LIN {X 0,Y 327.842,Z 1176.159,A -85,B 0,C 180,E1 13690.608,E2 13690.608} C_VEL
LIN {X 0,Y 330.278,Z 1159.38,A -85,B 0,C 180,E1 13695.569,E2 13695.569} C_VEL
LIN {X 0,Y 333.559,Z 1138.416,A -85,B 0,C 180,E1 13699.833,E2 13699.833} C_VEL
LIN {X 0,Y 337.656,Z 1111.754,A -85,B 0,C 180,E1 13703.592,E2 13703.592} C_VEL
LIN {X 0,Y 341.285,Z 1081.785,A -85,B 0,C 180,E1 13706.42,E2 13706.42} C_VEL
LIN {X 0,Y 343.694,Z 1048.536,A -85,B 0,C 180,E1 13708.37,E2 13708.37} C_VEL
LIN {X 0,Y 324.455,Z 997.109,A -85,B 0,C 180,E1 13712.143,E2 13712.143} C_VEL
LIN {X 0,Y 321.566,Z 989.03,A -85,B 0,C 180,E1 13712.907,E2 13712.907} C_VEL
LIN {X 0,Y 321.361,Z 989.03,A -85,B 0,C 180,E1 13715.329,E2 13715.329} C_VEL
LIN {X 0,Y 323.535,Z 994.456,A -85,B 0,C 180,E1 13716.08,E2 13716.08} C_VEL
LIN {X 0,Y 326.454,Z 998.467,A -85,B 0,C 180,E1 13716.933,E2 13716.933} C_VEL
LIN {X 0,Y 341.328,Z 1021.069,A -85,B 0,C 180,E1 13720.903,E2 13720.903} C_VEL
LIN {X 0,Y 357.405,Z 1050.395,A -85,B 0,C 180,E1 13724.791,E2 13724.791} C_VEL
LIN {X 0,Y 367.108,Z 1076.272,A -85,B 0,C 180,E1 13727.719,E2 13727.719} C_VEL
LIN {X 0,Y 361.475,Z 1112.177,A -85,B 0,C 180,E1 13729.868,E2 13729.868} C_VEL
LIN {X 0,Y 354.22,Z 1145.406,A -85,B 0,C 180,E1 13732.909,E2 13732.909} C_VEL
LIN {X 0,Y 346.259,Z 1175.129,A -85,B 0,C 180,E1 13736.799,E2 13736.799} C_VEL
LIN {X 0,Y 338.326,Z 1201.655,A -85,B 0,C 180,E1 13741.706,E2 13741.706} C_VEL
LIN {X 0,Y 331.825,Z 1222.692,A -85,B 0,C 180,E1 13747.254,E2 13747.254} C_VEL
LIN {X 0,Y 327.378,Z 1238.391,A -85,B 0,C 180,E1 13753.251,E2 13753.251} C_VEL
LIN {X 0,Y 325.075,Z 1248.624,A -85,B 0,C 180,E1 13759.294,E2 13759.294} C_VEL
LIN {X 0,Y 324.228,Z 1253.714,A -85,B 0,C 180,E1 13764.654,E2 13764.654} C_VEL
LIN {X 0,Y 323.952,Z 1255.427,A -85,B 0,C 180,E1 13769.995,E2 13769.995} C_VEL
LIN {X 0,Y 324.317,Z 1252.709,A -85,B 0,C 180,E1 13776.675,E2 13776.675} C_VEL
LIN {X 0,Y 325.921,Z 1244.536,A -85,B 0,C 180,E1 13783.38,E2 13783.38} C_VEL
LIN {X 0,Y 329.451,Z 1230.706,A -85,B 0,C 180,E1 13789.903,E2 13789.903} C_VEL
LIN {X 0,Y 335.08,Z 1211.817,A -85,B 0,C 180,E1 13795.758,E2 13795.758} C_VEL
LIN {X 0,Y 342.404,Z 1188.224,A -85,B 0,C 180,E1 13800.886,E2 13800.886} C_VEL
LIN {X 0,Y 350.57,Z 1159.61,A -85,B 0,C 180,E1 13805.301,E2 13805.301} C_VEL
LIN {X 0,Y 358.19,Z 1128.049,A -85,B 0,C 180,E1 13808.714,E2 13808.714} C_VEL
LIN {X 0,Y 364.641,Z 1093.639,A -85,B 0,C 180,E1 13811.261,E2 13811.261} C_VEL
LIN {X 0,Y 366.791,Z 1074.45,A -85,B 0,C 180,E1 13812.336,E2 13812.336} C_VEL
LIN {X 0,Y 354.759,Z 1045.172,A -85,B 0,C 180,E1 13815.748,E2 13815.748} C_VEL
LIN {X 0,Y 336.902,Z 1013.596,A -85,B 0,C 180,E1 13820.109,E2 13820.109} C_VEL
LIN {X 0,Y 323.813,Z 994.624,A -85,B 0,C 180,E1 13823.712,E2 13823.712} C_VEL
LIN {X 0,Y 321.462,Z 989.03,A -85,B 0,C 180,E1 13824.571,E2 13824.571} C_VEL
LIN {X 0,Y 321.795,Z 989.03,A -85,B 0,C 180,E1 13832.988,E2 13832.988} C_VEL
LIN {X 0,Y 322.198,Z 989.03,A -85,B 0,C 180,E1 13840.864,E2 13840.864} C_VEL
LIN {X 0,Y 322.712,Z 989.03,A -85,B 0,C 180,E1 13849.083,E2 13849.083} C_VEL
LIN {X 0,Y 323.215,Z 989.03,A -85,B 0,C 180,E1 13857.325,E2 13857.325} C_VEL
LIN {X 0,Y 323.277,Z 989.03,A -85,B 0,C 180,E1 13862.676,E2 13862.676} C_VEL
LIN {X 0,Y 322.641,Z 989.03,A -85,B 0,C 180,E1 13870.851,E2 13870.851} C_VEL
LIN {X 0,Y 322.111,Z 989.03,A -85,B 0,C 180,E1 13879.143,E2 13879.143} C_VEL
LIN {X 0,Y 321.771,Z 989.03,A -85,B 0,C 180,E1 13887.003,E2 13887.003} C_VEL
LIN {X 0,Y 321.635,Z 989.591,A -85,B 0,C 180,E1 13892.594,E2 13892.594} C_VEL
LIN {X 0,Y 326.494,Z 1001.003,A -85,B 0,C 180,E1 13894.238,E2 13894.238} C_VEL
LIN {X 0,Y 349.905,Z 1049.922,A -85,B 0,C 180,E1 13899.619,E2 13899.619} C_VEL
LIN {X 0,Y 364.312,Z 1087.174,A -85,B 0,C 180,E1 13903.441,E2 13903.441} C_VEL
LIN {X 0,Y 365.005,Z 1093.61,A -85,B 0,C 180,E1 13903.961,E2 13903.961} C_VEL
LIN {X 0,Y 357.243,Z 1134.418,A -85,B 0,C 180,E1 13906.643,E2 13906.643} C_VEL
LIN {X 0,Y 348.266,Z 1174.72,A -85,B 0,C 180,E1 13910.507,E2 13910.507} C_VEL
LIN {X 0,Y 340.072,Z 1213.611,A -85,B 0,C 180,E1 13915.375,E2 13915.375} C_VEL
LIN {X 0,Y 333.762,Z 1242.406,A -85,B 0,C 180,E1 13920.448,E2 13920.448} C_VEL
LIN {X 0,Y 328.614,Z 1266.532,A -85,B 0,C 180,E1 13926.32,E2 13926.32} C_VEL
LIN {X 0,Y 325.489,Z 1284.698,A -85,B 0,C 180,E1 13932.645,E2 13932.645} C_VEL
LIN {X 0,Y 324.33,Z 1296.014,A -85,B 0,C 180,E1 13938.468,E2 13938.468} C_VEL
LIN {X 0,Y 323.881,Z 1302.925,A -85,B 0,C 180,E1 13944.658,E2 13944.658} C_VEL
LIN {X 0,Y 323.958,Z 1304.876,A -85,B 0,C 180,E1 13950.005,E2 13950.005} C_VEL
LIN {X 0,Y 323.912,Z 1302.924,A -85,B 0,C 180,E1 13955.352,E2 13955.352} C_VEL
LIN {X 0,Y 324.362,Z 1295.959,A -85,B 0,C 180,E1 13961.572,E2 13961.572} C_VEL
LIN {X 0,Y 325.988,Z 1282.805,A -85,B 0,C 180,E1 13968.159,E2 13968.159} C_VEL
LIN {X 0,Y 329.344,Z 1264.057,A -85,B 0,C 180,E1 13974.36,E2 13974.36} C_VEL
LIN {X 0,Y 334.543,Z 1240.153,A -85,B 0,C 180,E1 13980.001,E2 13980.001} C_VEL
LIN {X 0,Y 338.144,Z 1224.571,A -85,B 0,C 180,E1 13982.848,E2 13982.848} C_VEL
LIN {X 0,Y 337.312,Z 1212.87,A -85,B 0,C 180,E1 13985.069,E2 13985.069} C_VEL
LIN {X 0,Y 336.399,Z 1202.111,A -85,B 0,C 180,E1 13986.93,E2 13986.93} C_VEL
LIN {X 0,Y 336.725,Z 1200.392,A -85,B 0,C 180,E1 13987.157,E2 13987.157} C_VEL
LIN {X 0,Y 343.446,Z 1167.637,A -85,B 0,C 180,E1 13990.804,E2 13990.804} C_VEL
LIN {X 0,Y 350.339,Z 1129.054,A -85,B 0,C 180,E1 13993.983,E2 13993.983} C_VEL
LIN {X 0,Y 360.86,Z 1090.849,A -85,B 0,C 180,E1 13997.195,E2 13997.195} C_VEL
LIN {X 0,Y 364.072,Z 1066.549,A -85,B 0,C 180,E1 14000.478,E2 14000.478} C_VEL
LIN {X 0,Y 363.409,Z 1063.296,A -85,B 0,C 180,E1 14002.097,E2 14002.097} C_VEL
LIN {X 0,Y 362.843,Z 1064.438,A -85,B 0,C 180,E1 14004.393,E2 14004.393} C_VEL
LIN {X 0,Y 359.681,Z 1073.138,A -85,B 0,C 180,E1 14005.221,E2 14005.221} C_VEL
LIN {X 0,Y 348.848,Z 1111.499,A -85,B 0,C 180,E1 14008.576,E2 14008.576} C_VEL
LIN {X 0,Y 341.201,Z 1138.326,A -85,B 0,C 180,E1 14012.044,E2 14012.044} C_VEL
LIN {X 0,Y 333.916,Z 1160.821,A -85,B 0,C 180,E1 14016.355,E2 14016.355} C_VEL
LIN {X 0,Y 327.641,Z 1177.723,A -85,B 0,C 180,E1 14021.192,E2 14021.192} C_VEL
LIN {X 0,Y 323.111,Z 1189.142,A -85,B 0,C 180,E1 14026.496,E2 14026.496} C_VEL
LIN {X 0,Y 320.196,Z 1195.188,A -85,B 0,C 180,E1 14031.872,E2 14031.872} C_VEL
LIN {X 0,Y 318.796,Z 1196.308,A -85,B 0,C 180,E1 14037.287,E2 14037.287} C_VEL
LIN {X 0,Y 318.677,Z 1192.532,A -85,B 0,C 180,E1 14042.713,E2 14042.713} C_VEL
LIN {X 0,Y 319.227,Z 1183.709,A -85,B 0,C 180,E1 14048.152,E2 14048.152} C_VEL
LIN {X 0,Y 321.312,Z 1168.881,A -85,B 0,C 180,E1 14053.58,E2 14053.58} C_VEL
LIN {X 0,Y 324.532,Z 1148.483,A -85,B 0,C 180,E1 14058.523,E2 14058.523} C_VEL
LIN {X 0,Y 328.668,Z 1122.896,A -85,B 0,C 180,E1 14062.74,E2 14062.74} C_VEL
LIN {X 0,Y 332.615,Z 1094.968,A -85,B 0,C 180,E1 14065.89,E2 14065.89} C_VEL
LIN {X 0,Y 335.845,Z 1063.866,A -85,B 0,C 180,E1 14068.183,E2 14068.183} C_VEL
LIN {X 0,Y 336.162,Z 1049.341,A -85,B 0,C 180,E1 14068.96,E2 14068.96} C_VEL
LIN {X 0,Y 316.792,Z 997.606,A -85,B 0,C 180,E1 14072.918,E2 14072.918} C_VEL
LIN {X 0,Y 314.162,Z 991.943,A -85,B 0,C 180,E1 14073.524,E2 14073.524} C_VEL
LIN {X 0,Y 318.931,Z 999.004,A -85,B 0,C 180,E1 14075.089,E2 14075.089} C_VEL
LIN {X 0,Y 333.802,Z 1021.018,A -85,B 0,C 180,E1 14079.365,E2 14079.365} C_VEL
LIN {X 0,Y 350.514,Z 1050.918,A -85,B 0,C 180,E1 14083.64,E2 14083.64} C_VEL
LIN {X 0,Y 361.022,Z 1078.194,A -85,B 0,C 180,E1 14086.924,E2 14086.924} C_VEL
LIN {X 0,Y 355.102,Z 1114.621,A -85,B 0,C 180,E1 14089.197,E2 14089.197} C_VEL
LIN {X 0,Y 347.376,Z 1148.214,A -85,B 0,C 180,E1 14092.376,E2 14092.376} C_VEL
LIN {X 0,Y 338.737,Z 1178.747,A -85,B 0,C 180,E1 14096.538,E2 14096.538} C_VEL
LIN {X 0,Y 330.839,Z 1203.66,A -85,B 0,C 180,E1 14101.378,E2 14101.378} C_VEL
LIN {X 0,Y 324.163,Z 1224.334,A -85,B 0,C 180,E1 14107.048,E2 14107.048} C_VEL
LIN {X 0,Y 319.393,Z 1240.43,A -85,B 0,C 180,E1 14113.526,E2 14113.526} C_VEL
LIN {X 0,Y 316.955,Z 1250.823,A -85,B 0,C 180,E1 14120.402,E2 14120.402} C_VEL
LIN {X 0,Y 316.173,Z 1255.575,A -85,B 0,C 180,E1 14127.259,E2 14127.259} C_VEL
LIN {X 0,Y 316.198,Z 1255.54,A -85,B 0,C 180,E1 14132.73,E2 14132.73} C_VEL
LIN {X 0,Y 316.945,Z 1250.727,A -85,B 0,C 180,E1 14139.587,E2 14139.587} C_VEL
LIN {X 0,Y 319.447,Z 1240.258,A -85,B 0,C 180,E1 14146.46,E2 14146.46} C_VEL
LIN {X 0,Y 324.215,Z 1224.067,A -85,B 0,C 180,E1 14152.937,E2 14152.937} C_VEL
LIN {X 0,Y 330.892,Z 1203.309,A -85,B 0,C 180,E1 14158.605,E2 14158.605} C_VEL
LIN {X 0,Y 339.197,Z 1177.241,A -85,B 0,C 180,E1 14163.59,E2 14163.59} C_VEL
LIN {X 0,Y 347.536,Z 1147.512,A -85,B 0,C 180,E1 14167.597,E2 14167.597} C_VEL
LIN {X 0,Y 354.85,Z 1115.563,A -85,B 0,C 180,E1 14170.625,E2 14170.625} C_VEL
LIN {X 0,Y 360.985,Z 1078.194,A -85,B 0,C 180,E1 14172.972,E2 14172.972} C_VEL
LIN {X 0,Y 349.196,Z 1048.427,A -85,B 0,C 180,E1 14176.591,E2 14176.591} C_VEL
LIN {X 0,Y 332.009,Z 1018.103,A -85,B 0,C 180,E1 14180.992,E2 14180.992} C_VEL
LIN {X 0,Y 316.548,Z 995.18,A -85,B 0,C 180,E1 14185.552,E2 14185.552} C_VEL
LIN {X 0,Y 313.63,Z 990.188,A -85,B 0,C 180,E1 14186.555,E2 14186.555} C_VEL
LIN {X 0,Y 313.543,Z 989.03,A -85,B 0,C 180,E1 14186.73,E2 14186.73} C_VEL
LIN {X 0,Y 313.9,Z 989.03,A -85,B 0,C 180,E1 14194.366,E2 14194.366} C_VEL
LIN {X 0,Y 314.252,Z 989.03,A -85,B 0,C 180,E1 14200.36,E2 14200.36} C_VEL
LIN {X 0,Y 314.623,Z 989.03,A -85,B 0,C 180,E1 14206.126,E2 14206.126} C_VEL
LIN {X 0,Y 315.194,Z 989.03,A -85,B 0,C 180,E1 14214.506,E2 14214.506} C_VEL
LIN {X 0,Y 315.547,Z 989.03,A -85,B 0,C 180,E1 14220.001,E2 14220.001} C_VEL
LIN {X 0,Y 314.913,Z 989.03,A -85,B 0,C 180,E1 14228.265,E2 14228.265} C_VEL
LIN {X 0,Y 314.348,Z 989.03,A -85,B 0,C 180,E1 14236.74,E2 14236.74} C_VEL
LIN {X 0,Y 313.896,Z 989.03,A -85,B 0,C 180,E1 14244.03,E2 14244.03} C_VEL
LIN {X 0,Y 313.713,Z 989.516,A -85,B 0,C 180,E1 14251.427,E2 14251.427} C_VEL
LIN {X 0,Y 321.069,Z 1005.61,A -85,B 0,C 180,E1 14253.62,E2 14253.62} C_VEL
LIN {X 0,Y 342.911,Z 1051.628,A -85,B 0,C 180,E1 14258.834,E2 14258.834} C_VEL
LIN {X 0,Y 357.162,Z 1088.674,A -85,B 0,C 180,E1 14262.792,E2 14262.792} C_VEL
LIN {X 0,Y 358.136,Z 1095.156,A -85,B 0,C 180,E1 14263.365,E2 14263.365} C_VEL
LIN {X 0,Y 350.166,Z 1135.277,A -85,B 0,C 180,E1 14266.092,E2 14266.092} C_VEL
LIN {X 0,Y 338.301,Z 1190.611,A -85,B 0,C 180,E1 14271.565,E2 14271.565} C_VEL
LIN {X 0,Y 331.425,Z 1221.512,A -85,B 0,C 180,E1 14275.929,E2 14275.929} C_VEL
LIN {X 0,Y 324.948,Z 1248.483,A -85,B 0,C 180,E1 14281.203,E2 14281.203} C_VEL
LIN {X 0,Y 320.163,Z 1270.395,A -85,B 0,C 180,E1 14287.128,E2 14287.128} C_VEL
LIN {X 0,Y 317.357,Z 1286.85,A -85,B 0,C 180,E1 14293.428,E2 14293.428} C_VEL
LIN {X 0,Y 316.362,Z 1296.606,A -85,B 0,C 180,E1 14299.006,E2 14299.006} C_VEL
LIN {X 0,Y 316.012,Z 1302.321,A -85,B 0,C 180,E1 14304.525,E2 14304.525} C_VEL
LIN {X 0,Y 316.104,Z 1304.276,A -85,B 0,C 180,E1 14310.005,E2 14310.005} C_VEL
LIN {X 0,Y 316.042,Z 1302.321,A -85,B 0,C 180,E1 14315.485,E2 14315.485} C_VEL
LIN {X 0,Y 316.51,Z 1295.348,A -85,B 0,C 180,E1 14321.863,E2 14321.863} C_VEL
LIN {X 0,Y 318.19,Z 1282.521,A -85,B 0,C 180,E1 14328.475,E2 14328.475} C_VEL
LIN {X 0,Y 321.855,Z 1263.434,A -85,B 0,C 180,E1 14334.965,E2 14334.965} C_VEL
LIN {X 0,Y 327.182,Z 1240.622,A -85,B 0,C 180,E1 14340.493,E2 14340.493} C_VEL
LIN {X 0,Y 333.928,Z 1212.709,A -85,B 0,C 180,E1 14345.43,E2 14345.43} C_VEL
LIN {X 0,Y 336.725,Z 1200.392,A -85,B 0,C 180,E1 14347.157,E2 14347.157} C_VEL
LIN {X 0,Y 336.432,Z 1187.381,A -85,B 0,C 180,E1 14349.14,E2 14349.14} C_VEL
LIN {X 0,Y 336.001,Z 1173.826,A -85,B 0,C 180,E1 14351.05,E2 14351.05} C_VEL
LIN {X 0,Y 343.866,Z 1132.971,A -85,B 0,C 180,E1 14354.607,E2 14354.607} C_VEL
LIN {X 0,Y 356.018,Z 1093.556,A -85,B 0,C 180,E1 14358.141,E2 14358.141} C_VEL
LIN {X 0,Y 360.214,Z 1071.69,A -85,B 0,C 180,E1 14361.386,E2 14361.386} C_VEL
LIN {X 0,Y 359.528,Z 1070.736,A -85,B 0,C 180,E1 14362.899,E2 14362.899} C_VEL
LIN {X 0,Y 358.958,Z 1072.007,A -85,B 0,C 180,E1 14363.79,E2 14363.79} C_VEL
LIN {X 0,Y 346.824,Z 1105.191,A -85,B 0,C 180,E1 14366.682,E2 14366.682} C_VEL
LIN {X 0,Y 337.416,Z 1135.219,A -85,B 0,C 180,E1 14370.348,E2 14370.348} C_VEL
LIN {X 0,Y 329.312,Z 1158.383,A -85,B 0,C 180,E1 14374.559,E2 14374.559} C_VEL
LIN {X 0,Y 321.97,Z 1176.979,A -85,B 0,C 180,E1 14379.632,E2 14379.632} C_VEL
LIN {X 0,Y 316.713,Z 1188.932,A -85,B 0,C 180,E1 14384.808,E2 14384.808} C_VEL
LIN {X 0,Y 313.197,Z 1195.941,A -85,B 0,C 180,E1 14390.292,E2 14390.292} C_VEL
LIN {X 0,Y 311.7,Z 1197.938,A -85,B 0,C 180,E1 14394.443,E2 14394.443} C_VEL
LIN {X 0,Y 310.898,Z 1196.392,A -85,B 0,C 180,E1 14399.999,E2 14399.999} C_VEL
LIN {X 0,Y 311.072,Z 1189.934,A -85,B 0,C 180,E1 14405.567,E2 14405.567} C_VEL
LIN {X 0,Y 312.428,Z 1178.022,A -85,B 0,C 180,E1 14411.138,E2 14411.138} C_VEL
LIN {X 0,Y 315.168,Z 1160.215,A -85,B 0,C 180,E1 14416.483,E2 14416.483} C_VEL
LIN {X 0,Y 319.063,Z 1137.233,A -85,B 0,C 180,E1 14421.137,E2 14421.137} C_VEL
LIN {X 0,Y 323.293,Z 1110.729,A -85,B 0,C 180,E1 14424.838,E2 14424.838} C_VEL
LIN {X 0,Y 327.037,Z 1081.274,A -85,B 0,C 180,E1 14427.627,E2 14427.627} C_VEL
LIN {X 0,Y 329.022,Z 1051.34,A -85,B 0,C 180,E1 14429.465,E2 14429.465} C_VEL
LIN {X 0,Y 311.515,Z 1003.891,A -85,B 0,C 180,E1 14433.272,E2 14433.272} C_VEL
LIN {X 0,Y 315.033,Z 1004.213,A -85,B 0,C 180,E1 14434.262,E2 14434.262} C_VEL
LIN {X 0,Y 331.258,Z 1029.023,A -85,B 0,C 180,E1 14439.092,E2 14439.092} C_VEL
LIN {X 0,Y 346.122,Z 1056.913,A -85,B 0,C 180,E1 14443.149,E2 14443.149} C_VEL
LIN {X 0,Y 355.015,Z 1080.978,A -85,B 0,C 180,E1 14446.161,E2 14446.161} C_VEL
LIN {X 0,Y 348.772,Z 1117.031,A -85,B 0,C 180,E1 14448.5,E2 14448.5} C_VEL
LIN {X 0,Y 340.844,Z 1149.896,A -85,B 0,C 180,E1 14451.69,E2 14451.69} C_VEL
LIN {X 0,Y 332.129,Z 1179.342,A -85,B 0,C 180,E1 14455.781,E2 14455.781} C_VEL
LIN {X 0,Y 323.86,Z 1204.261,A -85,B 0,C 180,E1 14460.702,E2 14460.702} C_VEL
LIN {X 0,Y 316.806,Z 1224.941,A -85,B 0,C 180,E1 14466.483,E2 14466.483} C_VEL
LIN {X 0,Y 311.778,Z 1241.034,A -85,B 0,C 180,E1 14473.112,E2 14473.112} C_VEL
LIN {X 0,Y 309.158,Z 1251.426,A -85,B 0,C 180,E1 14480.158,E2 14480.158} C_VEL
LIN {X 0,Y 308.296,Z 1256.177,A -85,B 0,C 180,E1 14487.189,E2 14487.189} C_VEL
LIN {X 0,Y 308.321,Z 1256.143,A -85,B 0,C 180,E1 14492.8,E2 14492.8} C_VEL
LIN {X 0,Y 309.148,Z 1251.331,A -85,B 0,C 180,E1 14499.832,E2 14499.832} C_VEL
LIN {X 0,Y 311.823,Z 1240.866,A -85,B 0,C 180,E1 14506.874,E2 14506.874} C_VEL
LIN {X 0,Y 316.875,Z 1224.676,A -85,B 0,C 180,E1 14513.5,E2 14513.5} C_VEL
LIN {X 0,Y 323.917,Z 1203.915,A -85,B 0,C 180,E1 14519.28,E2 14519.28} C_VEL
LIN {X 0,Y 332.594,Z 1177.843,A -85,B 0,C 180,E1 14524.349,E2 14524.349} C_VEL
LIN {X 0,Y 340.996,Z 1149.242,A -85,B 0,C 180,E1 14528.278,E2 14528.278} C_VEL
LIN {X 0,Y 348.514,Z 1117.987,A -85,B 0,C 180,E1 14531.318,E2 14531.318} C_VEL
LIN {X 0,Y 354.838,Z 1082.755,A -85,B 0,C 180,E1 14533.623,E2 14533.623} C_VEL
LIN {X 0,Y 350.86,Z 1068.778,A -85,B 0,C 180,E1 14535.233,E2 14535.233} C_VEL
LIN {X 0,Y 337.118,Z 1039.09,A -85,B 0,C 180,E1 14539.23,E2 14539.23} C_VEL
LIN {X 0,Y 321.388,Z 1013.578,A -85,B 0,C 180,E1 14543.601,E2 14543.601} C_VEL
LIN {X 0,Y 308.804,Z 995.31,A -85,B 0,C 180,E1 14547.738,E2 14547.738} C_VEL
LIN {X 0,Y 305.784,Z 990.191,A -85,B 0,C 180,E1 14548.892,E2 14548.892} C_VEL
LIN {X 0,Y 305.682,Z 989.03,A -85,B 0,C 180,E1 14549.13,E2 14549.13} C_VEL
LIN {X 0,Y 306.069,Z 989.03,A -85,B 0,C 180,E1 14556.772,E2 14556.772} C_VEL
LIN {X 0,Y 306.464,Z 989.03,A -85,B 0,C 180,E1 14562.818,E2 14562.818} C_VEL
LIN {X 0,Y 306.878,Z 989.03,A -85,B 0,C 180,E1 14569.544,E2 14569.544} C_VEL
LIN {X 0,Y 307.406,Z 989.03,A -85,B 0,C 180,E1 14577.187,E2 14577.187} C_VEL
LIN {X 0,Y 307.45,Z 989.03,A -85,B 0,C 180,E1 14582.814,E2 14582.814} C_VEL
LIN {X 0,Y 306.79,Z 989.03,A -85,B 0,C 180,E1 14591.347,E2 14591.347} C_VEL
LIN {X 0,Y 306.362,Z 989.03,A -85,B 0,C 180,E1 14597.189,E2 14597.189} C_VEL
LIN {X 0,Y 306.035,Z 989.03,A -85,B 0,C 180,E1 14603.232,E2 14603.232} C_VEL
LIN {X 0,Y 305.787,Z 989.513,A -85,B 0,C 180,E1 14610.217,E2 14610.217} C_VEL
LIN {X 0,Y 331.983,Z 1044.448,A -85,B 0,C 180,E1 14617.031,E2 14617.031} C_VEL
LIN {X 0,Y 347.243,Z 1082.028,A -85,B 0,C 180,E1 14621.241,E2 14621.241} C_VEL
LIN {X 0,Y 351.243,Z 1096.676,A -85,B 0,C 180,E1 14622.751,E2 14622.751} C_VEL
LIN {X 0,Y 342.748,Z 1137.423,A -85,B 0,C 180,E1 14625.652,E2 14625.652} C_VEL
LIN {X 0,Y 333.546,Z 1182.943,A -85,B 0,C 180,E1 14629.863,E2 14629.863} C_VEL
LIN {X 0,Y 325.934,Z 1215.257,A -85,B 0,C 180,E1 14634.194,E2 14634.194} C_VEL
LIN {X 0,Y 318.997,Z 1243.26,A -85,B 0,C 180,E1 14639.439,E2 14639.439} C_VEL
LIN {X 0,Y 313.317,Z 1266.602,A -85,B 0,C 180,E1 14645.534,E2 14645.534} C_VEL
LIN {X 0,Y 309.911,Z 1284.212,A -85,B 0,C 180,E1 14652.087,E2 14652.087} C_VEL
LIN {X 0,Y 308.491,Z 1295.994,A -85,B 0,C 180,E1 14658.722,E2 14658.722} C_VEL
LIN {X 0,Y 308.125,Z 1301.717,A -85,B 0,C 180,E1 14664.384,E2 14664.384} C_VEL
LIN {X 0,Y 308.223,Z 1303.675,A -85,B 0,C 180,E1 14670.005,E2 14670.005} C_VEL
LIN {X 0,Y 308.157,Z 1301.717,A -85,B 0,C 180,E1 14675.626,E2 14675.626} C_VEL
LIN {X 0,Y 308.634,Z 1294.852,A -85,B 0,C 180,E1 14682.088,E2 14682.088} C_VEL
LIN {X 0,Y 310.433,Z 1281.899,A -85,B 0,C 180,E1 14688.954,E2 14688.954} C_VEL
LIN {X 0,Y 314.423,Z 1262.813,A -85,B 0,C 180,E1 14695.597,E2 14695.597} C_VEL
LIN {X 0,Y 320.459,Z 1238.681,A -85,B 0,C 180,E1 14701.523,E2 14701.523} C_VEL
LIN {X 0,Y 328.063,Z 1208.903,A -85,B 0,C 180,E1 14706.732,E2 14706.732} C_VEL
LIN {X 0,Y 335.108,Z 1178.061,A -85,B 0,C 180,E1 14710.602,E2 14710.602} C_VEL
LIN {X 0,Y 336.001,Z 1173.826,A -85,B 0,C 180,E1 14711.05,E2 14711.05} C_VEL
LIN {X 0,Y 335.675,Z 1159.744,A -85,B 0,C 180,E1 14712.836,E2 14712.836} C_VEL
LIN {X 0,Y 335.217,Z 1145.107,A -85,B 0,C 180,E1 14714.475,E2 14714.475} C_VEL
LIN {X 0,Y 351.463,Z 1096.768,A -85,B 0,C 180,E1 14719.077,E2 14719.077} C_VEL
LIN {X 0,Y 356.158,Z 1079.085,A -85,B 0,C 180,E1 14721.765,E2 14721.765} C_VEL
LIN {X 0,Y 356.283,Z 1077.707,A -85,B 0,C 180,E1 14722.503,E2 14722.503} C_VEL
LIN {X 0,Y 355.21,Z 1079.638,A -85,B 0,C 180,E1 14723.024,E2 14723.024} C_VEL
LIN {X 0,Y 341.927,Z 1110.917,A -85,B 0,C 180,E1 14725.95,E2 14725.95} C_VEL
LIN {X 0,Y 331.015,Z 1140.662,A -85,B 0,C 180,E1 14729.904,E2 14729.904} C_VEL
LIN {X 0,Y 322.199,Z 1163.055,A -85,B 0,C 180,E1 14734.329,E2 14734.329} C_VEL
LIN {X 0,Y 314.207,Z 1181.108,A -85,B 0,C 180,E1 14739.732,E2 14739.732} C_VEL
LIN {X 0,Y 308.819,Z 1192.227,A -85,B 0,C 180,E1 14745.136,E2 14745.136} C_VEL
LIN {X 0,Y 304.94,Z 1198.663,A -85,B 0,C 180,E1 14751.462,E2 14751.462} C_VEL
LIN {X 0,Y 303.291,Z 1199.279,A -85,B 0,C 180,E1 14757.148,E2 14757.148} C_VEL
LIN {X 0,Y 303.129,Z 1195.033,A -85,B 0,C 180,E1 14762.853,E2 14762.853} C_VEL
LIN {X 0,Y 303.729,Z 1185.751,A -85,B 0,C 180,E1 14768.571,E2 14768.571} C_VEL
LIN {X 0,Y 306,Z 1170.426,A -85,B 0,C 180,E1 14774.273,E2 14774.273} C_VEL
LIN {X 0,Y 309.383,Z 1150.525,A -85,B 0,C 180,E1 14779.221,E2 14779.221} C_VEL
LIN {X 0,Y 313.685,Z 1125.705,A -85,B 0,C 180,E1 14783.496,E2 14783.496} C_VEL
LIN {X 0,Y 318.151,Z 1096.182,A -85,B 0,C 180,E1 14786.97,E2 14786.97} C_VEL
LIN {X 0,Y 321.584,Z 1064.723,A -85,B 0,C 180,E1 14789.348,E2 14789.348} C_VEL
LIN {X 0,Y 321.721,Z 1053,A -85,B 0,C 180,E1 14790.026,E2 14790.026} C_VEL
LIN {X 0,Y 308.683,Z 1016.372,A -85,B 0,C 180,E1 14792.983,E2 14792.983} C_VEL
LIN {X 0,Y 311.839,Z 1014.491,A -85,B 0,C 180,E1 14793.801,E2 14793.801} C_VEL
LIN {X 0,Y 313.367,Z 1013.169,A -85,B 0,C 180,E1 14794.169,E2 14794.169} C_VEL
LIN {X 0,Y 328.804,Z 1037.171,A -85,B 0,C 180,E1 14798.836,E2 14798.836} C_VEL
LIN {X 0,Y 342.124,Z 1063.999,A -85,B 0,C 180,E1 14802.803,E2 14802.803} C_VEL
LIN {X 0,Y 349.015,Z 1084.747,A -85,B 0,C 180,E1 14805.46,E2 14805.46} C_VEL
LIN {X 0,Y 342.8,Z 1118.038,A -85,B 0,C 180,E1 14807.661,E2 14807.661} C_VEL
LIN {X 0,Y 334.676,Z 1150.479,A -85,B 0,C 180,E1 14810.85,E2 14810.85} C_VEL
LIN {X 0,Y 325.491,Z 1180.21,A -85,B 0,C 180,E1 14815.042,E2 14815.042} C_VEL
LIN {X 0,Y 316.426,Z 1206.264,A -85,B 0,C 180,E1 14820.338,E2 14820.338} C_VEL
LIN {X 0,Y 309.176,Z 1226.582,A -85,B 0,C 180,E1 14826.249,E2 14826.249} C_VEL
LIN {X 0,Y 304.146,Z 1241.641,A -85,B 0,C 180,E1 14832.675,E2 14832.675} C_VEL
LIN {X 0,Y 301.346,Z 1252.03,A -85,B 0,C 180,E1 14839.9,E2 14839.9} C_VEL
LIN {X 0,Y 300.42,Z 1256.779,A -85,B 0,C 180,E1 14847.115,E2 14847.115} C_VEL
LIN {X 0,Y 300.472,Z 1256.743,A -85,B 0,C 180,E1 14852.873,E2 14852.873} C_VEL
LIN {X 0,Y 301.336,Z 1251.936,A -85,B 0,C 180,E1 14860.089,E2 14860.089} C_VEL
LIN {X 0,Y 304.193,Z 1241.475,A -85,B 0,C 180,E1 14867.311,E2 14867.311} C_VEL
LIN {X 0,Y 309.595,Z 1225.282,A -85,B 0,C 180,E1 14874.087,E2 14874.087} C_VEL
LIN {X 0,Y 317.013,Z 1204.518,A -85,B 0,C 180,E1 14879.982,E2 14879.982} C_VEL
LIN {X 0,Y 326.329,Z 1177.482,A -85,B 0,C 180,E1 14885.297,E2 14885.297} C_VEL
LIN {X 0,Y 335.33,Z 1147.972,A -85,B 0,C 180,E1 14889.334,E2 14889.334} C_VEL
LIN {X 0,Y 343.293,Z 1115.609,A -85,B 0,C 180,E1 14892.431,E2 14892.431} C_VEL
LIN {X 0,Y 348.883,Z 1083.239,A -85,B 0,C 180,E1 14894.572,E2 14894.572} C_VEL
LIN {X 0,Y 337.721,Z 1054.232,A -85,B 0,C 180,E1 14898.455,E2 14898.455} C_VEL
LIN {X 0,Y 322.216,Z 1026.167,A -85,B 0,C 180,E1 14902.935,E2 14902.935} C_VEL
LIN {X 0,Y 305.9,Z 1002.075,A -85,B 0,C 180,E1 14908.323,E2 14908.323} C_VEL
LIN {X 0,Y 300.89,Z 995.243,A -85,B 0,C 180,E1 14910.259,E2 14910.259} C_VEL
LIN {X 0,Y 297.968,Z 990.481,A -85,B 0,C 180,E1 14911.515,E2 14911.515} C_VEL
LIN {X 0,Y 297.819,Z 989.03,A -85,B 0,C 180,E1 14911.854,E2 14911.854} C_VEL
LIN {X 0,Y 298.27,Z 989.03,A -85,B 0,C 180,E1 14919.261,E2 14919.261} C_VEL
LIN {X 0,Y 298.7,Z 989.03,A -85,B 0,C 180,E1 14925.37,E2 14925.37} C_VEL
LIN {X 0,Y 299.321,Z 989.03,A -85,B 0,C 180,E1 14934.214,E2 14934.214} C_VEL
LIN {X 0,Y 299.737,Z 989.03,A -85,B 0,C 180,E1 14940.001,E2 14940.001} C_VEL
LIN {X 0,Y 299.259,Z 989.03,A -85,B 0,C 180,E1 14945.788,E2 14945.788} C_VEL
LIN {X 0,Y 298.827,Z 989.03,A -85,B 0,C 180,E1 14951.653,E2 14951.653} C_VEL
LIN {X 0,Y 298.394,Z 989.03,A -85,B 0,C 180,E1 14957.663,E2 14957.663} C_VEL
LIN {X 0,Y 297.972,Z 989.03,A -85,B 0,C 180,E1 14964.287,E2 14964.287} C_VEL
LIN {X 0,Y 297.906,Z 989.71,A -85,B 0,C 180,E1 14967.563,E2 14967.563} C_VEL
LIN {X 0,Y 300.321,Z 994.801,A -85,B 0,C 180,E1 14968.663,E2 14968.663} C_VEL
LIN {X 0,Y 303.063,Z 997.786,A -85,B 0,C 180,E1 14969.72,E2 14969.72} C_VEL
LIN {X 0,Y 311.119,Z 1016.517,A -85,B 0,C 180,E1 14972.593,E2 14972.593} C_VEL
LIN {X 0,Y 330.409,Z 1058.548,A -85,B 0,C 180,E1 14977.643,E2 14977.643} C_VEL
LIN {X 0,Y 344.211,Z 1096.059,A -85,B 0,C 180,E1 14981.954,E2 14981.954} C_VEL
LIN {X 0,Y 331.104,Z 1164.506,A -85,B 0,C 180,E1 14987.101,E2 14987.101} C_VEL
LIN {X 0,Y 323.646,Z 1197.495,A -85,B 0,C 180,E1 14990.81,E2 14990.81} C_VEL
LIN {X 0,Y 315.922,Z 1227.693,A -85,B 0,C 180,E1 14995.593,E2 14995.593} C_VEL
LIN {X 0,Y 308.962,Z 1253.518,A -85,B 0,C 180,E1 15001.31,E2 15001.31} C_VEL
LIN {X 0,Y 303.975,Z 1274.312,A -85,B 0,C 180,E1 15007.763,E2 15007.763} C_VEL
LIN {X 0,Y 301.268,Z 1289.787,A -85,B 0,C 180,E1 15014.759,E2 15014.759} C_VEL
LIN {X 0,Y 300.373,Z 1298.777,A -85,B 0,C 180,E1 15021.337,E2 15021.337} C_VEL
LIN {X 0,Y 300.22,Z 1302.543,A -85,B 0,C 180,E1 15027.124,E2 15027.124} C_VEL
LIN {X 0,Y 300.254,Z 1302.544,A -85,B 0,C 180,E1 15032.886,E2 15032.886} C_VEL
LIN {X 0,Y 300.378,Z 1298.775,A -85,B 0,C 180,E1 15038.674,E2 15038.674} C_VEL
LIN {X 0,Y 301.326,Z 1289.781,A -85,B 0,C 180,E1 15045.249,E2 15045.249} C_VEL
LIN {X 0,Y 304.159,Z 1274.321,A -85,B 0,C 180,E1 15052.235,E2 15052.235} C_VEL
LIN {X 0,Y 309.368,Z 1253.363,A -85,B 0,C 180,E1 15058.713,E2 15058.713} C_VEL
LIN {X 0,Y 316.451,Z 1227.443,A -85,B 0,C 180,E1 15064.418,E2 15064.418} C_VEL
LIN {X 0,Y 324.259,Z 1197.408,A -85,B 0,C 180,E1 15069.141,E2 15069.141} C_VEL
LIN {X 0,Y 331.674,Z 1164.609,A -85,B 0,C 180,E1 15072.821,E2 15072.821} C_VEL
LIN {X 0,Y 335.217,Z 1145.107,A -85,B 0,C 180,E1 15074.475,E2 15074.475} C_VEL
LIN {X 0,Y 337.236,Z 1134.616,A -85,B 0,C 180,E1 15075.779,E2 15075.779} C_VEL
LIN {X 0,Y 339.599,Z 1119.626,A -85,B 0,C 180,E1 15078.222,E2 15078.222} C_VEL
LIN {X 0,Y 339.936,Z 1118.739,A -85,B 0,C 180,E1 15078.315,E2 15078.315} C_VEL
LIN {X 0,Y 347.478,Z 1099.49,A -85,B 0,C 180,E1 15080.163,E2 15080.163} C_VEL
LIN {X 0,Y 351.701,Z 1087.161,A -85,B 0,C 180,E1 15082.173,E2 15082.173} C_VEL
LIN {X 0,Y 335.693,Z 1120.201,A -85,B 0,C 180,E1 15085.619,E2 15085.619} C_VEL
LIN {X 0,Y 324.114,Z 1147.585,A -85,B 0,C 180,E1 15089.705,E2 15089.705} C_VEL
LIN {X 0,Y 313.995,Z 1170.159,A -85,B 0,C 180,E1 15094.754,E2 15094.754} C_VEL
LIN {X 0,Y 305.611,Z 1186.764,A -85,B 0,C 180,E1 15100.532,E2 15100.532} C_VEL
LIN {X 0,Y 300.919,Z 1195.318,A -85,B 0,C 180,E1 15105.479,E2 15105.479} C_VEL
LIN {X 0,Y 297.34,Z 1200.432,A -85,B 0,C 180,E1 15111.242,E2 15111.242} C_VEL
LIN {X 0,Y 295.545,Z 1200.769,A -85,B 0,C 180,E1 15117.073,E2 15117.073} C_VEL
LIN {X 0,Y 295.349,Z 1196.269,A -85,B 0,C 180,E1 15122.928,E2 15122.928} C_VEL
LIN {X 0,Y 295.993,Z 1186.721,A -85,B 0,C 180,E1 15128.797,E2 15128.797} C_VEL
LIN {X 0,Y 298.381,Z 1171.103,A -85,B 0,C 180,E1 15134.646,E2 15134.646} C_VEL
LIN {X 0,Y 301.917,Z 1150.912,A -85,B 0,C 180,E1 15139.715,E2 15139.715} C_VEL
LIN {X 0,Y 306.551,Z 1124.818,A -85,B 0,C 180,E1 15144.221,E2 15144.221} C_VEL
LIN {X 0,Y 311.045,Z 1095.598,A -85,B 0,C 180,E1 15147.638,E2 15147.638} C_VEL
LIN {X 0,Y 314.66,Z 1062.959,A -85,B 0,C 180,E1 15150.08,E2 15150.08} C_VEL
LIN {X 0,Y 314.262,Z 1054.071,A -85,B 0,C 180,E1 15150.646,E2 15150.646} C_VEL
LIN {X 0,Y 305.796,Z 1029.361,A -85,B 0,C 180,E1 15152.691,E2 15152.691} C_VEL
LIN {X 0,Y 308.795,Z 1027.615,A -85,B 0,C 180,E1 15153.488,E2 15153.488} C_VEL
LIN {X 0,Y 310.904,Z 1023.642,A -85,B 0,C 180,E1 15153.917,E2 15153.917} C_VEL
LIN {X 0,Y 313.721,Z 1024.866,A -85,B 0,C 180,E1 15154.734,E2 15154.734} C_VEL
LIN {X 0,Y 328.591,Z 1049.817,A -85,B 0,C 180,E1 15159.311,E2 15159.311} C_VEL
LIN {X 0,Y 340.337,Z 1077.405,A -85,B 0,C 180,E1 15163.368,E2 15163.368} C_VEL
LIN {X 0,Y 343.102,Z 1087.449,A -85,B 0,C 180,E1 15164.659,E2 15164.659} C_VEL
LIN {X 0,Y 336.691,Z 1120.015,A -85,B 0,C 180,E1 15166.875,E2 15166.875} C_VEL
LIN {X 0,Y 327.813,Z 1153.756,A -85,B 0,C 180,E1 15170.297,E2 15170.297} C_VEL
LIN {X 0,Y 318.307,Z 1182.763,A -85,B 0,C 180,E1 15174.574,E2 15174.574} C_VEL
LIN {X 0,Y 309.018,Z 1208.267,A -85,B 0,C 180,E1 15179.958,E2 15179.958} C_VEL
LIN {X 0,Y 301.186,Z 1229.152,A -85,B 0,C 180,E1 15186.364,E2 15186.364} C_VEL
LIN {X 0,Y 296.139,Z 1243.514,A -85,B 0,C 180,E1 15192.956,E2 15192.956} C_VEL
LIN {X 0,Y 293.555,Z 1252.633,A -85,B 0,C 180,E1 15199.629,E2 15199.629} C_VEL
LIN {X 0,Y 292.543,Z 1257.38,A -85,B 0,C 180,E1 15207.037,E2 15207.037} C_VEL
LIN {X 0,Y 292.595,Z 1257.345,A -85,B 0,C 180,E1 15212.951,E2 15212.951} C_VEL
LIN {X 0,Y 293.546,Z 1252.541,A -85,B 0,C 180,E1 15220.36,E2 15220.36} C_VEL
LIN {X 0,Y 296.596,Z 1242.083,A -85,B 0,C 180,E1 15227.769,E2 15227.769} C_VEL
LIN {X 0,Y 302.32,Z 1225.891,A -85,B 0,C 180,E1 15234.705,E2 15234.705} C_VEL
LIN {X 0,Y 310.138,Z 1205.124,A -85,B 0,C 180,E1 15240.718,E2 15240.718} C_VEL
LIN {X 0,Y 319.746,Z 1178.507,A -85,B 0,C 180,E1 15246.049,E2 15246.049} C_VEL
LIN {X 0,Y 329.141,Z 1148.931,A -85,B 0,C 180,E1 15250.164,E2 15250.164} C_VEL
LIN {X 0,Y 337.663,Z 1115.476,A -85,B 0,C 180,E1 15253.396,E2 15253.396} C_VEL
LIN {X 0,Y 342.821,Z 1085.637,A -85,B 0,C 180,E1 15255.428,E2 15255.428} C_VEL
LIN {X 0,Y 332.094,Z 1057.165,A -85,B 0,C 180,E1 15259.435,E2 15259.435} C_VEL
LIN {X 0,Y 317.486,Z 1030.497,A -85,B 0,C 180,E1 15263.933,E2 15263.933} C_VEL
LIN {X 0,Y 302.625,Z 1008.322,A -85,B 0,C 180,E1 15269.073,E2 15269.073} C_VEL
LIN {X 0,Y 297.161,Z 1001.038,A -85,B 0,C 180,E1 15271.275,E2 15271.275} C_VEL
LIN {X 0,Y 293.657,Z 995.698,A -85,B 0,C 180,E1 15272.856,E2 15272.856} C_VEL
LIN {X 0,Y 290.276,Z 991.145,A -85,B 0,C 180,E1 15274.474,E2 15274.474} C_VEL
LIN {X 0,Y 290.003,Z 989.03,A -85,B 0,C 180,E1 15274.987,E2 15274.987} C_VEL
LIN {X 0,Y 290.486,Z 989.03,A -85,B 0,C 180,E1 15281.841,E2 15281.841} C_VEL
LIN {X 0,Y 291.031,Z 989.03,A -85,B 0,C 180,E1 15290.093,E2 15290.093} C_VEL
LIN {X 0,Y 291.6,Z 989.03,A -85,B 0,C 180,E1 15297.034,E2 15297.034} C_VEL
LIN {X 0,Y 291.631,Z 989.03,A -85,B 0,C 180,E1 15302.966,E2 15302.966} C_VEL
LIN {X 0,Y 290.865,Z 989.03,A -85,B 0,C 180,E1 15311.977,E2 15311.977} C_VEL
LIN {X 0,Y 290.297,Z 989.03,A -85,B 0,C 180,E1 15320.675,E2 15320.675} C_VEL
LIN {X 0,Y 290.07,Z 989.64,A -85,B 0,C 180,E1 15324.491,E2 15324.491} C_VEL
LIN {X 0,Y 292.355,Z 994.689,A -85,B 0,C 180,E1 15325.714,E2 15325.714} C_VEL
LIN {X 0,Y 295.308,Z 997.747,A -85,B 0,C 180,E1 15327.016,E2 15327.016} C_VEL
LIN {X 0,Y 300.851,Z 1006.115,A -85,B 0,C 180,E1 15329.38,E2 15329.38} C_VEL
LIN {X 0,Y 312.455,Z 1035.245,A -85,B 0,C 180,E1 15333.762,E2 15333.762} C_VEL
LIN {X 0,Y 329.658,Z 1076.191,A -85,B 0,C 180,E1 15338.763,E2 15338.763} C_VEL
LIN {X 0,Y 337.323,Z 1099.807,A -85,B 0,C 180,E1 15341.523,E2 15341.523} C_VEL
LIN {X 0,Y 326.777,Z 1156.578,A -85,B 0,C 180,E1 15345.476,E2 15345.476} C_VEL
LIN {X 0,Y 319.37,Z 1189.196,A -85,B 0,C 180,E1 15348.884,E2 15348.884} C_VEL
LIN {X 0,Y 310.922,Z 1220.65,A -85,B 0,C 180,E1 15353.556,E2 15353.556} C_VEL
LIN {X 0,Y 303.561,Z 1246.604,A -85,B 0,C 180,E1 15358.958,E2 15358.958} C_VEL
LIN {X 0,Y 297.615,Z 1268.501,A -85,B 0,C 180,E1 15365.278,E2 15365.278} C_VEL
LIN {X 0,Y 294.115,Z 1284.994,A -85,B 0,C 180,E1 15372.076,E2 15372.076} C_VEL
LIN {X 0,Y 292.768,Z 1295.049,A -85,B 0,C 180,E1 15378.315,E2 15378.315} C_VEL
LIN {X 0,Y 292.358,Z 1300.507,A -85,B 0,C 180,E1 15384.08,E2 15384.08} C_VEL
LIN {X 0,Y 292.473,Z 1302.473,A -85,B 0,C 180,E1 15390.006,E2 15390.006} C_VEL
LIN {X 0,Y 292.389,Z 1300.509,A -85,B 0,C 180,E1 15395.931,E2 15395.931} C_VEL
LIN {X 0,Y 292.889,Z 1293.752,A -85,B 0,C 180,E1 15402.655,E2 15402.655} C_VEL
LIN {X 0,Y 294.816,Z 1281.639,A -85,B 0,C 180,E1 15409.522,E2 15409.522} C_VEL
LIN {X 0,Y 299.338,Z 1262.935,A -85,B 0,C 180,E1 15416.544,E2 15416.544} C_VEL
LIN {X 0,Y 306.151,Z 1238.764,A -85,B 0,C 180,E1 15422.84,E2 15422.84} C_VEL
LIN {X 0,Y 314.237,Z 1210.719,A -85,B 0,C 180,E1 15428.058,E2 15428.058} C_VEL
LIN {X 0,Y 322.478,Z 1178.725,A -85,B 0,C 180,E1 15432.282,E2 15432.282} C_VEL
LIN {X 0,Y 330.612,Z 1143.135,A -85,B 0,C 180,E1 15435.736,E2 15435.736} C_VEL
LIN {X 0,Y 339.936,Z 1118.739,A -85,B 0,C 180,E1 15438.315,E2 15438.315} C_VEL
LIN {X 0,Y 342.194,Z 1110.397,A -85,B 0,C 180,E1 15439.645,E2 15439.645} C_VEL
LIN {X 0,Y 343.978,Z 1102.993,A -85,B 0,C 180,E1 15441.205,E2 15441.205} C_VEL
LIN {X 0,Y 345.258,Z 1099.586,A -85,B 0,C 180,E1 15441.875,E2 15441.875} C_VEL
LIN {X 0,Y 328.985,Z 1129.846,A -85,B 0,C 180,E1 15445.417,E2 15445.417} C_VEL
LIN {X 0,Y 316.182,Z 1156.246,A -85,B 0,C 180,E1 15449.927,E2 15449.927} C_VEL
LIN {X 0,Y 305.757,Z 1176.753,A -85,B 0,C 180,E1 15455.197,E2 15455.197} C_VEL
LIN {X 0,Y 297.776,Z 1190.664,A -85,B 0,C 180,E1 15460.768,E2 15460.768} C_VEL
LIN {X 0,Y 292.454,Z 1199.088,A -85,B 0,C 180,E1 15466.574,E2 15466.574} C_VEL
LIN {X 0,Y 289.026,Z 1202.717,A -85,B 0,C 180,E1 15472.803,E2 15472.803} C_VEL
LIN {X 0,Y 287.796,Z 1202.259,A -85,B 0,C 180,E1 15476.994,E2 15476.994} C_VEL
LIN {X 0,Y 287.582,Z 1197.488,A -85,B 0,C 180,E1 15483.007,E2 15483.007} C_VEL
LIN {X 0,Y 288.259,Z 1187.682,A -85,B 0,C 180,E1 15489.035,E2 15489.035} C_VEL
LIN {X 0,Y 290.755,Z 1171.709,A -85,B 0,C 180,E1 15495.039,E2 15495.039} C_VEL
LIN {X 0,Y 294.45,Z 1151.215,A -85,B 0,C 180,E1 15500.237,E2 15500.237} C_VEL
LIN {X 0,Y 299.206,Z 1125.281,A -85,B 0,C 180,E1 15504.779,E2 15504.779} C_VEL
LIN {X 0,Y 303.749,Z 1096.814,A -85,B 0,C 180,E1 15508.159,E2 15508.159} C_VEL
LIN {X 0,Y 307.523,Z 1063.785,A -85,B 0,C 180,E1 15510.687,E2 15510.687} C_VEL
LIN {X 0,Y 307.097,Z 1055.948,A -85,B 0,C 180,E1 15511.212,E2 15511.212} C_VEL
LIN {X 0,Y 303.03,Z 1042.793,A -85,B 0,C 180,E1 15512.451,E2 15512.451} C_VEL
LIN {X 0,Y 306.22,Z 1040.275,A -85,B 0,C 180,E1 15513.282,E2 15513.282} C_VEL
LIN {X 0,Y 309.365,Z 1035.438,A -85,B 0,C 180,E1 15513.973,E2 15513.973} C_VEL
LIN {X 0,Y 311.881,Z 1033.265,A -85,B 0,C 180,E1 15514.576,E2 15514.576} C_VEL
LIN {X 0,Y 326.404,Z 1059.596,A -85,B 0,C 180,E1 15519.36,E2 15519.36} C_VEL
LIN {X 0,Y 336.538,Z 1086.742,A -85,B 0,C 180,E1 15523.396,E2 15523.396} C_VEL
LIN {X 0,Y 336.8,Z 1092.695,A -85,B 0,C 180,E1 15523.967,E2 15523.967} C_VEL
LIN {X 0,Y 329.263,Z 1127.711,A -85,B 0,C 180,E1 15526.563,E2 15526.563} C_VEL
LIN {X 0,Y 320.159,Z 1159.275,A -85,B 0,C 180,E1 15530.037,E2 15530.037} C_VEL
LIN {X 0,Y 310.643,Z 1186.693,A -85,B 0,C 180,E1 15534.336,E2 15534.336} C_VEL
LIN {X 0,Y 301.093,Z 1211.596,A -85,B 0,C 180,E1 15539.915,E2 15539.915} C_VEL
LIN {X 0,Y 293.167,Z 1231.617,A -85,B 0,C 180,E1 15546.483,E2 15546.483} C_VEL
LIN {X 0,Y 288.104,Z 1245.389,A -85,B 0,C 180,E1 15553.251,E2 15553.251} C_VEL
LIN {X 0,Y 285.422,Z 1254.662,A -85,B 0,C 180,E1 15560.868,E2 15560.868} C_VEL
LIN {X 0,Y 284.686,Z 1257.98,A -85,B 0,C 180,E1 15566.956,E2 15566.956} C_VEL
LIN {X 0,Y 284.73,Z 1257.946,A -85,B 0,C 180,E1 15573.032,E2 15573.032} C_VEL
LIN {X 0,Y 285.749,Z 1253.146,A -85,B 0,C 180,E1 15580.646,E2 15580.646} C_VEL
LIN {X 0,Y 289.025,Z 1242.69,A -85,B 0,C 180,E1 15588.25,E2 15588.25} C_VEL
LIN {X 0,Y 295.097,Z 1226.498,A -85,B 0,C 180,E1 15595.352,E2 15595.352} C_VEL
LIN {X 0,Y 303.311,Z 1205.73,A -85,B 0,C 180,E1 15601.487,E2 15601.487} C_VEL
LIN {X 0,Y 313,Z 1180.182,A -85,B 0,C 180,E1 15606.724,E2 15606.724} C_VEL
LIN {X 0,Y 322.696,Z 1151.024,A -85,B 0,C 180,E1 15610.89,E2 15610.89} C_VEL
LIN {X 0,Y 331.204,Z 1119.393,A -85,B 0,C 180,E1 15614.049,E2 15614.049} C_VEL
LIN {X 0,Y 337.139,Z 1089.233,A -85,B 0,C 180,E1 15616.154,E2 15616.154} C_VEL
LIN {X 0,Y 327.007,Z 1061.086,A -85,B 0,C 180,E1 15620.298,E2 15620.298} C_VEL
LIN {X 0,Y 312.345,Z 1033.733,A -85,B 0,C 180,E1 15625.142,E2 15625.142} C_VEL
LIN {X 0,Y 296.238,Z 1009.603,A -85,B 0,C 180,E1 15631.177,E2 15631.177} C_VEL
LIN {X 0,Y 290.365,Z 1002.043,A -85,B 0,C 180,E1 15633.821,E2 15633.821} C_VEL
LIN {X 0,Y 286.355,Z 996.019,A -85,B 0,C 180,E1 15635.905,E2 15635.905} C_VEL
LIN {X 0,Y 282.659,Z 991.509,A -85,B 0,C 180,E1 15637.98,E2 15637.98} C_VEL
LIN {X 0,Y 282.319,Z 989.03,A -85,B 0,C 180,E1 15638.429,E2 15638.429} C_VEL
LIN {X 0,Y 282.748,Z 989.03,A -85,B 0,C 180,E1 15644.525,E2 15644.525} C_VEL
LIN {X 0,Y 283.286,Z 989.03,A -85,B 0,C 180,E1 15652.948,E2 15652.948} C_VEL
LIN {X 0,Y 283.926,Z 989.03,A -85,B 0,C 180,E1 15660.001,E2 15660.001} C_VEL
LIN {X 0,Y 283.388,Z 989.03,A -85,B 0,C 180,E1 15666.114,E2 15666.114} C_VEL
LIN {X 0,Y 282.895,Z 989.03,A -85,B 0,C 180,E1 15672.32,E2 15672.32} C_VEL
LIN {X 0,Y 282.386,Z 989.665,A -85,B 0,C 180,E1 15680.891,E2 15680.891} C_VEL
LIN {X 0,Y 284.558,Z 994.605,A -85,B 0,C 180,E1 15682.302,E2 15682.302} C_VEL
LIN {X 0,Y 287.626,Z 997.529,A -85,B 0,C 180,E1 15683.893,E2 15683.893} C_VEL
LIN {X 0,Y 291.827,Z 1003.22,A -85,B 0,C 180,E1 15685.968,E2 15685.968} C_VEL
LIN {X 0,Y 297.837,Z 1012.602,A -85,B 0,C 180,E1 15688.668,E2 15688.668} C_VEL
LIN {X 0,Y 318.563,Z 1067.654,A -85,B 0,C 180,E1 15696.728,E2 15696.728} C_VEL
LIN {X 0,Y 330.219,Z 1100.526,A -85,B 0,C 180,E1 15700.799,E2 15700.799} C_VEL
LIN {X 0,Y 323.492,Z 1143.759,A -85,B 0,C 180,E1 15703.458,E2 15703.458} C_VEL
LIN {X 0,Y 315.705,Z 1178.646,A -85,B 0,C 180,E1 15706.701,E2 15706.701} C_VEL
LIN {X 0,Y 307.19,Z 1210.469,A -85,B 0,C 180,E1 15711.012,E2 15711.012} C_VEL
LIN {X 0,Y 298.927,Z 1238.103,A -85,B 0,C 180,E1 15716.275,E2 15716.275} C_VEL
LIN {X 0,Y 291.819,Z 1262.167,A -85,B 0,C 180,E1 15722.687,E2 15722.687} C_VEL
LIN {X 0,Y 287.377,Z 1279.564,A -85,B 0,C 180,E1 15729.247,E2 15729.247} C_VEL
LIN {X 0,Y 285.14,Z 1292.126,A -85,B 0,C 180,E1 15736.228,E2 15736.228} C_VEL
LIN {X 0,Y 284.552,Z 1298.842,A -85,B 0,C 180,E1 15742.387,E2 15742.387} C_VEL
LIN {X 0,Y 284.45,Z 1301.337,A -85,B 0,C 180,E1 15746.965,E2 15746.965} C_VEL
LIN {X 0,Y 284.48,Z 1301.339,A -85,B 0,C 180,E1 15753.047,E2 15753.047} C_VEL
LIN {X 0,Y 284.621,Z 1297.559,A -85,B 0,C 180,E1 15759.158,E2 15759.158} C_VEL
LIN {X 0,Y 285.717,Z 1288.548,A -85,B 0,C 180,E1 15766.104,E2 15766.104} C_VEL
LIN {X 0,Y 289.026,Z 1273.192,A -85,B 0,C 180,E1 15773.421,E2 15773.421} C_VEL
LIN {X 0,Y 294.603,Z 1253.505,A -85,B 0,C 180,E1 15779.868,E2 15779.868} C_VEL
LIN {X 0,Y 302.574,Z 1227.709,A -85,B 0,C 180,E1 15785.882,E2 15785.882} C_VEL
LIN {X 0,Y 311.302,Z 1197.714,A -85,B 0,C 180,E1 15790.837,E2 15790.837} C_VEL
LIN {X 0,Y 319.585,Z 1164.994,A -85,B 0,C 180,E1 15794.646,E2 15794.646} C_VEL
LIN {X 0,Y 323.836,Z 1149.034,A -85,B 0,C 180,E1 15796.249,E2 15796.249} C_VEL
LIN {X 0,Y 343.978,Z 1102.993,A -85,B 0,C 180,E1 15801.205,E2 15801.205} C_VEL
LIN {X 0,Y 343.187,Z 1103.463,A -85,B 0,C 180,E1 15801.864,E2 15801.864} C_VEL
LIN {X 0,Y 338.848,Z 1110.482,A -85,B 0,C 180,E1 15802.667,E2 15802.667} C_VEL
LIN {X 0,Y 328.565,Z 1127.896,A -85,B 0,C 180,E1 15803.608,E2 15803.608} C_VEL
LIN {X 0,Y 327.279,Z 1130.054,A -85,B 0,C 180,E1 15803.871,E2 15803.871} C_VEL
LIN {X 0,Y 312.34,Z 1156.802,A -85,B 0,C 180,E1 15808.464,E2 15808.464} C_VEL
LIN {X 0,Y 300.407,Z 1177.838,A -85,B 0,C 180,E1 15813.927,E2 15813.927} C_VEL
LIN {X 0,Y 291.596,Z 1191.866,A -85,B 0,C 180,E1 15819.555,E2 15819.555} C_VEL
LIN {X 0,Y 285.049,Z 1201.155,A -85,B 0,C 180,E1 15826.218,E2 15826.218} C_VEL
LIN {X 0,Y 282.162,Z 1204.006,A -85,B 0,C 180,E1 15830.767,E2 15830.767} C_VEL
LIN {X 0,Y 280.05,Z 1203.735,A -85,B 0,C 180,E1 15836.911,E2 15836.911} C_VEL
LIN {X 0,Y 279.802,Z 1198.68,A -85,B 0,C 180,E1 15843.091,E2 15843.091} C_VEL
LIN {X 0,Y 280.495,Z 1188.559,A -85,B 0,C 180,E1 15849.287,E2 15849.287} C_VEL
LIN {X 0,Y 283.131,Z 1172.316,A -85,B 0,C 180,E1 15855.454,E2 15855.454} C_VEL
LIN {X 0,Y 287.007,Z 1151.471,A -85,B 0,C 180,E1 15860.786,E2 15860.786} C_VEL
LIN {X 0,Y 291.801,Z 1126.119,A -85,B 0,C 180,E1 15865.275,E2 15865.275} C_VEL
LIN {X 0,Y 296.721,Z 1096.029,A -85,B 0,C 180,E1 15868.888,E2 15868.888} C_VEL
LIN {X 0,Y 300.564,Z 1063.393,A -85,B 0,C 180,E1 15871.392,E2 15871.392} C_VEL
LIN {X 0,Y 299.534,Z 1055.696,A -85,B 0,C 180,E1 15872.093,E2 15872.093} C_VEL
LIN {X 0,Y 302.892,Z 1053.413,A -85,B 0,C 180,E1 15872.98,E2 15872.98} C_VEL
LIN {X 0,Y 306.369,Z 1048.597,A -85,B 0,C 180,E1 15873.737,E2 15873.737} C_VEL
LIN {X 0,Y 310.644,Z 1042.915,A -85,B 0,C 180,E1 15874.636,E2 15874.636} C_VEL
LIN {X 0,Y 323.378,Z 1068.381,A -85,B 0,C 180,E1 15879.26,E2 15879.26} C_VEL
LIN {X 0,Y 331.257,Z 1091.515,A -85,B 0,C 180,E1 15882.806,E2 15882.806} C_VEL
LIN {X 0,Y 324.027,Z 1126.662,A -85,B 0,C 180,E1 15885.45,E2 15885.45} C_VEL
LIN {X 0,Y 314.545,Z 1158.637,A -85,B 0,C 180,E1 15888.947,E2 15888.947} C_VEL
LIN {X 0,Y 304.23,Z 1187.287,A -85,B 0,C 180,E1 15893.464,E2 15893.464} C_VEL
LIN {X 0,Y 294.213,Z 1212.198,A -85,B 0,C 180,E1 15899.135,E2 15899.135} C_VEL
LIN {X 0,Y 286.626,Z 1230.363,A -85,B 0,C 180,E1 15905.084,E2 15905.084} C_VEL
LIN {X 0,Y 280.921,Z 1244.727,A -85,B 0,C 180,E1 15912.002,E2 15912.002} C_VEL
LIN {X 0,Y 277.965,Z 1253.841,A -85,B 0,C 180,E1 15919.04,E2 15919.04} C_VEL
LIN {X 0,Y 276.81,Z 1258.582,A -85,B 0,C 180,E1 15926.869,E2 15926.869} C_VEL
LIN {X 0,Y 276.854,Z 1258.548,A -85,B 0,C 180,E1 15933.119,E2 15933.119} C_VEL
LIN {X 0,Y 277.957,Z 1253.752,A -85,B 0,C 180,E1 15940.948,E2 15940.948} C_VEL
LIN {X 0,Y 281.479,Z 1243.298,A -85,B 0,C 180,E1 15948.758,E2 15948.758} C_VEL
LIN {X 0,Y 287.842,Z 1227.222,A -85,B 0,C 180,E1 15955.993,E2 15955.993} C_VEL
LIN {X 0,Y 296.359,Z 1206.815,A -85,B 0,C 180,E1 15962.166,E2 15962.166} C_VEL
LIN {X 0,Y 306.884,Z 1180.179,A -85,B 0,C 180,E1 15967.713,E2 15967.713} C_VEL
LIN {X 0,Y 317.067,Z 1150.54,A -85,B 0,C 180,E1 15971.96,E2 15971.96} C_VEL
LIN {X 0,Y 326.328,Z 1116.813,A -85,B 0,C 180,E1 15975.287,E2 15975.287} C_VEL
LIN {X 0,Y 331.38,Z 1092.943,A -85,B 0,C 180,E1 15976.92,E2 15976.92} C_VEL
LIN {X 0,Y 322.524,Z 1066.474,A -85,B 0,C 180,E1 15980.94,E2 15980.94} C_VEL
LIN {X 0,Y 309.934,Z 1041.67,A -85,B 0,C 180,E1 15985.472,E2 15985.472} C_VEL
LIN {X 0,Y 293.923,Z 1016.742,A -85,B 0,C 180,E1 15991.656,E2 15991.656} C_VEL
LIN {X 0,Y 283.884,Z 1003.102,A -85,B 0,C 180,E1 15996.615,E2 15996.615} C_VEL
LIN {X 0,Y 280.113,Z 997.436,A -85,B 0,C 180,E1 15998.911,E2 15998.911} C_VEL
LIN {X 0,Y 274.97,Z 991.334,A -85,B 0,C 180,E1 16002.497,E2 16002.497} C_VEL
LIN {X 0,Y 274.667,Z 989.03,A -85,B 0,C 180,E1 16003.176,E2 16003.176} C_VEL
LIN {X 0,Y 275.273,Z 989.03,A -85,B 0,C 180,E1 16010.63,E2 16010.63} C_VEL
LIN {X 0,Y 275.754,Z 989.03,A -85,B 0,C 180,E1 16016.864,E2 16016.864} C_VEL
LIN {X 0,Y 275.796,Z 989.03,A -85,B 0,C 180,E1 16023.137,E2 16023.137} C_VEL
LIN {X 0,Y 275.192,Z 989.03,A -85,B 0,C 180,E1 16029.469,E2 16029.469} C_VEL
LIN {X 0,Y 274.666,Z 989.686,A -85,B 0,C 180,E1 16036.287,E2 16036.287} C_VEL
LIN {X 0,Y 276.757,Z 994.548,A -85,B 0,C 180,E1 16038.066,E2 16038.066} C_VEL
LIN {X 0,Y 280.172,Z 997.382,A -85,B 0,C 180,E1 16040.253,E2 16040.253} C_VEL
LIN {X 0,Y 284.049,Z 1003.168,A -85,B 0,C 180,E1 16042.603,E2 16042.603} C_VEL
LIN {X 0,Y 294.537,Z 1018.038,A -85,B 0,C 180,E1 16047.768,E2 16047.768} C_VEL
LIN {X 0,Y 314.668,Z 1074.327,A -85,B 0,C 180,E1 16056.188,E2 16056.188} C_VEL
LIN {X 0,Y 324.357,Z 1103.919,A -85,B 0,C 180,E1 16060.035,E2 16060.035} C_VEL
LIN {X 0,Y 318.456,Z 1141.024,A -85,B 0,C 180,E1 16062.241,E2 16062.241} C_VEL
LIN {X 0,Y 310.227,Z 1176.489,A -85,B 0,C 180,E1 16065.497,E2 16065.497} C_VEL
LIN {X 0,Y 300.96,Z 1209.49,A -85,B 0,C 180,E1 16069.966,E2 16069.966} C_VEL
LIN {X 0,Y 292.099,Z 1237.477,A -85,B 0,C 180,E1 16075.376,E2 16075.376} C_VEL
LIN {X 0,Y 284.509,Z 1261.539,A -85,B 0,C 180,E1 16081.925,E2 16081.925} C_VEL
LIN {X 0,Y 279.347,Z 1280.564,A -85,B 0,C 180,E1 16089.45,E2 16089.45} C_VEL
LIN {X 0,Y 277.176,Z 1292.528,A -85,B 0,C 180,E1 16096.627,E2 16096.627} C_VEL
LIN {X 0,Y 276.588,Z 1299.296,A -85,B 0,C 180,E1 16103.742,E2 16103.742} C_VEL
LIN {X 0,Y 276.732,Z 1301.272,A -85,B 0,C 180,E1 16110.006,E2 16110.006} C_VEL
LIN {X 0,Y 276.617,Z 1299.299,A -85,B 0,C 180,E1 16116.27,E2 16116.27} C_VEL
LIN {X 0,Y 277.22,Z 1292.527,A -85,B 0,C 180,E1 16123.383,E2 16123.383} C_VEL
LIN {X 0,Y 279.469,Z 1280.572,A -85,B 0,C 180,E1 16130.554,E2 16130.554} C_VEL
LIN {X 0,Y 284.376,Z 1262.783,A -85,B 0,C 180,E1 16137.673,E2 16137.673} C_VEL
LIN {X 0,Y 291.917,Z 1239.206,A -85,B 0,C 180,E1 16144.202,E2 16144.202} C_VEL
LIN {X 0,Y 300.803,Z 1211.553,A -85,B 0,C 180,E1 16149.639,E2 16149.639} C_VEL
LIN {X 0,Y 310.059,Z 1179.667,A -85,B 0,C 180,E1 16154.069,E2 16154.069} C_VEL
LIN {X 0,Y 316.534,Z 1156.068,A -85,B 0,C 180,E1 16156.646,E2 16156.646} C_VEL
LIN {X 0,Y 337.329,Z 1113.924,A -85,B 0,C 180,E1 16161.486,E2 16161.486} C_VEL
LIN {X 0,Y 337.517,Z 1113.285,A -85,B 0,C 180,E1 16161.771,E2 16161.771} C_VEL
LIN {X 0,Y 327.279,Z 1130.054,A -85,B 0,C 180,E1 16163.871,E2 16163.871} C_VEL
LIN {X 0,Y 310.78,Z 1154.792,A -85,B 0,C 180,E1 16166.386,E2 16166.386} C_VEL
LIN {X 0,Y 309.926,Z 1156.157,A -85,B 0,C 180,E1 16166.645,E2 16166.645} C_VEL
LIN {X 0,Y 296.001,Z 1178.146,A -85,B 0,C 180,E1 16172.278,E2 16172.278} C_VEL
LIN {X 0,Y 285.631,Z 1193.149,A -85,B 0,C 180,E1 16178.296,E2 16178.296} C_VEL
LIN {X 0,Y 278.961,Z 1201.792,A -85,B 0,C 180,E1 16184.308,E2 16184.308} C_VEL
LIN {X 0,Y 274.57,Z 1205.769,A -85,B 0,C 180,E1 16190.51,E2 16190.51} C_VEL
LIN {X 0,Y 272.301,Z 1205.17,A -85,B 0,C 180,E1 16196.823,E2 16196.823} C_VEL
LIN {X 0,Y 271.992,Z 1199.816,A -85,B 0,C 180,E1 16203.18,E2 16203.18} C_VEL
LIN {X 0,Y 272.734,Z 1189.41,A -85,B 0,C 180,E1 16209.553,E2 16209.553} C_VEL
LIN {X 0,Y 275.537,Z 1172.828,A -85,B 0,C 180,E1 16215.891,E2 16215.891} C_VEL
LIN {X 0,Y 279.597,Z 1151.688,A -85,B 0,C 180,E1 16221.363,E2 16221.363} C_VEL
LIN {X 0,Y 284.563,Z 1125.981,A -85,B 0,C 180,E1 16225.94,E2 16225.94} C_VEL
LIN {X 0,Y 289.468,Z 1096.967,A -85,B 0,C 180,E1 16229.469,E2 16229.469} C_VEL
LIN {X 0,Y 292.463,Z 1074.975,A -85,B 0,C 180,E1 16231.406,E2 16231.406} C_VEL
LIN {X 0,Y 296.238,Z 1071.497,A -85,B 0,C 180,E1 16232.307,E2 16232.307} C_VEL
LIN {X 0,Y 301.541,Z 1062.468,A -85,B 0,C 180,E1 16233.196,E2 16233.196} C_VEL
LIN {X 0,Y 309.71,Z 1053.573,A -85,B 0,C 180,E1 16234.922,E2 16234.922} C_VEL
LIN {X 0,Y 321.446,Z 1080.687,A -85,B 0,C 180,E1 16239.787,E2 16239.787} C_VEL
LIN {X 0,Y 325.578,Z 1096.342,A -85,B 0,C 180,E1 16242.125,E2 16242.125} C_VEL
LIN {X 0,Y 317.582,Z 1130.284,A -85,B 0,C 180,E1 16244.741,E2 16244.741} C_VEL
LIN {X 0,Y 307.768,Z 1161.673,A -85,B 0,C 180,E1 16248.31,E2 16248.31} C_VEL
LIN {X 0,Y 297.183,Z 1189.735,A -85,B 0,C 180,E1 16252.908,E2 16252.908} C_VEL
LIN {X 0,Y 286.828,Z 1214.074,A -85,B 0,C 180,E1 16258.692,E2 16258.692} C_VEL
LIN {X 0,Y 278.577,Z 1232.83,A -85,B 0,C 180,E1 16265.17,E2 16265.17} C_VEL
LIN {X 0,Y 272.883,Z 1246.6,A -85,B 0,C 180,E1 16272.286,E2 16272.286} C_VEL
LIN {X 0,Y 269.798,Z 1255.869,A -85,B 0,C 180,E1 16280.334,E2 16280.334} C_VEL
LIN {X 0,Y 268.934,Z 1259.184,A -85,B 0,C 180,E1 16286.777,E2 16286.777} C_VEL
LIN {X 0,Y 268.978,Z 1259.15,A -85,B 0,C 180,E1 16293.21,E2 16293.21} C_VEL
LIN {X 0,Y 270.172,Z 1254.404,A -85,B 0,C 180,E1 16301.215,E2 16301.215} C_VEL
LIN {X 0,Y 273.965,Z 1243.904,A -85,B 0,C 180,E1 16309.292,E2 16309.292} C_VEL
LIN {X 0,Y 280.933,Z 1227.278,A -85,B 0,C 180,E1 16316.91,E2 16316.91} C_VEL
LIN {X 0,Y 290.109,Z 1206.318,A -85,B 0,C 180,E1 16323.296,E2 16323.296} C_VEL
LIN {X 0,Y 300.846,Z 1180.248,A -85,B 0,C 180,E1 16328.728,E2 16328.728} C_VEL
LIN {X 0,Y 311.303,Z 1150.864,A -85,B 0,C 180,E1 16332.969,E2 16332.969} C_VEL
LIN {X 0,Y 320.838,Z 1117.396,A -85,B 0,C 180,E1 16336.286,E2 16336.286} C_VEL
LIN {X 0,Y 325.651,Z 1095.29,A -85,B 0,C 180,E1 16337.846,E2 16337.846} C_VEL
LIN {X 0,Y 316.293,Z 1067.597,A -85,B 0,C 180,E1 16342.321,E2 16342.321} C_VEL
LIN {X 0,Y 304.738,Z 1044.917,A -85,B 0,C 180,E1 16346.787,E2 16346.787} C_VEL
LIN {X 0,Y 290.85,Z 1023.084,A -85,B 0,C 180,E1 16352.482,E2 16352.482} C_VEL
LIN {X 0,Y 281.469,Z 1010.078,A -85,B 0,C 180,E1 16357.339,E2 16357.339} C_VEL
LIN {X 0,Y 276.768,Z 1003.345,A -85,B 0,C 180,E1 16360.372,E2 16360.372} C_VEL
LIN {X 0,Y 272.939,Z 997.833,A -85,B 0,C 180,E1 16363.335,E2 16363.335} C_VEL
LIN {X 0,Y 270.76,Z 995.824,A -85,B 0,C 180,E1 16365.211,E2 16365.211} C_VEL
LIN {X 0,Y 267.308,Z 990.463,A -85,B 0,C 180,E1 16369.224,E2 16369.224} C_VEL
LIN {X 0,Y 267.233,Z 989.03,A -85,B 0,C 180,E1 16369.837,E2 16369.837} C_VEL
LIN {X 0,Y 267.829,Z 989.03,A -85,B 0,C 180,E1 16376.771,E2 16376.771} C_VEL
LIN {X 0,Y 267.865,Z 989.03,A -85,B 0,C 180,E1 16383.23,E2 16383.23} C_VEL
LIN {X 0,Y 267.268,Z 989.687,A -85,B 0,C 180,E1 16389.752,E2 16389.752} C_VEL
LIN {X 0,Y 268.955,Z 994.214,A -85,B 0,C 180,E1 16392.146,E2 16392.146} C_VEL
LIN {X 0,Y 272.849,Z 997.616,A -85,B 0,C 180,E1 16395.717,E2 16395.717} C_VEL
LIN {X 0,Y 276.367,Z 1003.098,A -85,B 0,C 180,E1 16398.504,E2 16398.504} C_VEL
LIN {X 0,Y 278.509,Z 1005.689,A -85,B 0,C 180,E1 16399.938,E2 16399.938} C_VEL
LIN {X 0,Y 284.232,Z 1014.035,A -85,B 0,C 180,E1 16403.364,E2 16403.364} C_VEL
LIN {X 0,Y 291.505,Z 1024.186,A -85,B 0,C 180,E1 16406.959,E2 16406.959} C_VEL
LIN {X 0,Y 310.24,Z 1078.619,A -85,B 0,C 180,E1 16415.281,E2 16415.281} C_VEL
LIN {X 0,Y 318.764,Z 1107.248,A -85,B 0,C 180,E1 16419.123,E2 16419.123} C_VEL
LIN {X 0,Y 312.754,Z 1141.94,A -85,B 0,C 180,E1 16421.262,E2 16421.262} C_VEL
LIN {X 0,Y 304.191,Z 1176.928,A -85,B 0,C 180,E1 16424.54,E2 16424.54} C_VEL
LIN {X 0,Y 294.622,Z 1209.181,A -85,B 0,C 180,E1 16428.993,E2 16428.993} C_VEL
LIN {X 0,Y 285.287,Z 1236.846,A -85,B 0,C 180,E1 16434.426,E2 16434.426} C_VEL
LIN {X 0,Y 277.257,Z 1260.911,A -85,B 0,C 180,E1 16441.122,E2 16441.122} C_VEL
LIN {X 0,Y 271.723,Z 1279.942,A -85,B 0,C 180,E1 16448.846,E2 16448.846} C_VEL
LIN {X 0,Y 269.368,Z 1291.915,A -85,B 0,C 180,E1 16456.232,E2 16456.232} C_VEL
LIN {X 0,Y 268.707,Z 1298.691,A -85,B 0,C 180,E1 16463.557,E2 16463.557} C_VEL
LIN {X 0,Y 268.87,Z 1300.672,A -85,B 0,C 180,E1 16470.006,E2 16470.006} C_VEL
LIN {X 0,Y 268.734,Z 1298.694,A -85,B 0,C 180,E1 16476.455,E2 16476.455} C_VEL
LIN {X 0,Y 269.413,Z 1291.916,A -85,B 0,C 180,E1 16483.778,E2 16483.778} C_VEL
LIN {X 0,Y 271.836,Z 1279.951,A -85,B 0,C 180,E1 16491.158,E2 16491.158} C_VEL
LIN {X 0,Y 277.139,Z 1262.162,A -85,B 0,C 180,E1 16498.46,E2 16498.46} C_VEL
LIN {X 0,Y 285.163,Z 1238.588,A -85,B 0,C 180,E1 16505.13,E2 16505.13} C_VEL
LIN {X 0,Y 294.218,Z 1211.862,A -85,B 0,C 180,E1 16510.501,E2 16510.501} C_VEL
LIN {X 0,Y 304.189,Z 1179.34,A -85,B 0,C 180,E1 16515.105,E2 16515.105} C_VEL
LIN {X 0,Y 309.323,Z 1162.93,A -85,B 0,C 180,E1 16517.044,E2 16517.044} C_VEL
LIN {X 0,Y 329.268,Z 1126.752,A -85,B 0,C 180,E1 16521.779,E2 16521.779} C_VEL
LIN {X 0,Y 310.52,Z 1155.165,A -85,B 0,C 180,E1 16526.443,E2 16526.443} C_VEL
LIN {X 0,Y 309.926,Z 1156.157,A -85,B 0,C 180,E1 16526.645,E2 16526.645} C_VEL
LIN {X 0,Y 301.049,Z 1167.845,A -85,B 0,C 180,E1 16528.459,E2 16528.459} C_VEL
LIN {X 0,Y 293.018,Z 1177.283,A -85,B 0,C 180,E1 16530.19,E2 16530.19} C_VEL
LIN {X 0,Y 292.163,Z 1178.405,A -85,B 0,C 180,E1 16530.514,E2 16530.514} C_VEL
LIN {X 0,Y 279.791,Z 1194.664,A -85,B 0,C 180,E1 16537.083,E2 16537.083} C_VEL
LIN {X 0,Y 271.686,Z 1203.979,A -85,B 0,C 180,E1 16543.876,E2 16543.876} C_VEL
LIN {X 0,Y 266.993,Z 1207.549,A -85,B 0,C 180,E1 16550.238,E2 16550.238} C_VEL
LIN {X 0,Y 264.557,Z 1206.6,A -85,B 0,C 180,E1 16556.73,E2 16556.73} C_VEL
LIN {X 0,Y 264.199,Z 1200.937,A -85,B 0,C 180,E1 16563.274,E2 16563.274} C_VEL
LIN {X 0,Y 264.978,Z 1190.215,A -85,B 0,C 180,E1 16569.836,E2 16569.836} C_VEL
LIN {X 0,Y 267.938,Z 1173.334,A -85,B 0,C 180,E1 16576.354,E2 16576.354} C_VEL
LIN {X 0,Y 272.207,Z 1151.71,A -85,B 0,C 180,E1 16581.973,E2 16581.973} C_VEL
LIN {X 0,Y 277.679,Z 1124.28,A -85,B 0,C 180,E1 16586.853,E2 16586.853} C_VEL
LIN {X 0,Y 282.851,Z 1094.906,A -85,B 0,C 180,E1 16590.45,E2 16590.45} C_VEL
LIN {X 0,Y 286.333,Z 1092.563,A -85,B 0,C 180,E1 16591.358,E2 16591.358} C_VEL
LIN {X 0,Y 293.315,Z 1082.11,A -85,B 0,C 180,E1 16592.431,E2 16592.431} C_VEL
LIN {X 0,Y 300.075,Z 1073.791,A -85,B 0,C 180,E1 16593.69,E2 16593.69} C_VEL
LIN {X 0,Y 303.827,Z 1068.04,A -85,B 0,C 180,E1 16594.289,E2 16594.289} C_VEL
LIN {X 0,Y 308.025,Z 1063.907,A -85,B 0,C 180,E1 16595.141,E2 16595.141} C_VEL
LIN {X 0,Y 317.57,Z 1089.099,A -85,B 0,C 180,E1 16599.681,E2 16599.681} C_VEL
LIN {X 0,Y 319.681,Z 1099.946,A -85,B 0,C 180,E1 16601.275,E2 16601.275} C_VEL
LIN {X 0,Y 311.249,Z 1133.74,A -85,B 0,C 180,E1 16603.99,E2 16603.99} C_VEL
LIN {X 0,Y 300.608,Z 1165.903,A -85,B 0,C 180,E1 16607.815,E2 16607.815} C_VEL
LIN {X 0,Y 289.379,Z 1193.761,A -85,B 0,C 180,E1 16612.676,E2 16612.676} C_VEL
LIN {X 0,Y 278.875,Z 1217.227,A -85,B 0,C 180,E1 16618.605,E2 16618.605} C_VEL
LIN {X 0,Y 270.545,Z 1235.295,A -85,B 0,C 180,E1 16625.264,E2 16625.264} C_VEL
LIN {X 0,Y 264.415,Z 1249.517,A -85,B 0,C 180,E1 16633.413,E2 16633.413} C_VEL
LIN {X 0,Y 262.001,Z 1256.472,A -85,B 0,C 180,E1 16640.043,E2 16640.043} C_VEL
LIN {X 0,Y 261.059,Z 1259.786,A -85,B 0,C 180,E1 16646.68,E2 16646.68} C_VEL
LIN {X 0,Y 261.102,Z 1259.753,A -85,B 0,C 180,E1 16653.307,E2 16653.307} C_VEL
LIN {X 0,Y 262.298,Z 1255.311,A -85,B 0,C 180,E1 16661.211,E2 16661.211} C_VEL
LIN {X 0,Y 265.904,Z 1245.787,A -85,B 0,C 180,E1 16669.039,E2 16669.039} C_VEL
LIN {X 0,Y 272.921,Z 1229.911,A -85,B 0,C 180,E1 16676.899,E2 16676.899} C_VEL
LIN {X 0,Y 282.433,Z 1209.219,A -85,B 0,C 180,E1 16683.571,E2 16683.571} C_VEL
LIN {X 0,Y 293.498,Z 1183.845,A -85,B 0,C 180,E1 16689.16,E2 16689.16} C_VEL
LIN {X 0,Y 304.681,Z 1154.157,A -85,B 0,C 180,E1 16693.647,E2 16693.647} C_VEL
LIN {X 0,Y 314.397,Z 1121.956,A -85,B 0,C 180,E1 16696.981,E2 16696.981} C_VEL
LIN {X 0,Y 319.693,Z 1097.246,A -85,B 0,C 180,E1 16698.897,E2 16698.897} C_VEL
LIN {X 0,Y 310.577,Z 1069.835,A -85,B 0,C 180,E1 16703.584,E2 16703.584} C_VEL
LIN {X 0,Y 299.219,Z 1047.159,A -85,B 0,C 180,E1 16708.347,E2 16708.347} C_VEL
LIN {X 0,Y 286.764,Z 1027.837,A -85,B 0,C 180,E1 16713.855,E2 16713.855} C_VEL
LIN {X 0,Y 279.114,Z 1016.945,A -85,B 0,C 180,E1 16718.076,E2 16718.076} C_VEL
LIN {X 0,Y 274.83,Z 1010.621,A -85,B 0,C 180,E1 16720.975,E2 16720.975} C_VEL
LIN {X 0,Y 271.019,Z 1004.461,A -85,B 0,C 180,E1 16724.132,E2 16724.132} C_VEL
LIN {X 0,Y 266.194,Z 998.997,A -85,B 0,C 180,E1 16729.281,E2 16729.281} C_VEL
LIN {X 0,Y 265.737,Z 996.775,A -85,B 0,C 180,E1 16730.193,E2 16730.193} C_VEL
LIN {X 0,Y 262.592,Z 994.885,A -85,B 0,C 180,E1 16741.647,E2 16741.647} C_VEL
LIN {X 0,Y 265.871,Z 997.616,A -85,B 0,C 180,E1 16749.25,E2 16749.25} C_VEL
LIN {X 0,Y 268.91,Z 1003.138,A -85,B 0,C 180,E1 16753.135,E2 16753.135} C_VEL
LIN {X 0,Y 271.29,Z 1005.487,A -85,B 0,C 180,E1 16755.307,E2 16755.307} C_VEL
LIN {X 0,Y 275.436,Z 1011.103,A -85,B 0,C 180,E1 16758.569,E2 16758.569} C_VEL
LIN {X 0,Y 285.797,Z 1026.215,A -85,B 0,C 180,E1 16764.779,E2 16764.779} C_VEL
LIN {X 0,Y 289.209,Z 1032.438,A -85,B 0,C 180,E1 16766.514,E2 16766.514} C_VEL
LIN {X 0,Y 306.493,Z 1085.289,A -85,B 0,C 180,E1 16774.699,E2 16774.699} C_VEL
LIN {X 0,Y 313.217,Z 1110.379,A -85,B 0,C 180,E1 16778.176,E2 16778.176} C_VEL
LIN {X 0,Y 306.466,Z 1145.904,A -85,B 0,C 180,E1 16780.485,E2 16780.485} C_VEL
LIN {X 0,Y 297.08,Z 1181.362,A -85,B 0,C 180,E1 16784.023,E2 16784.023} C_VEL
LIN {X 0,Y 286.982,Z 1212.831,A -85,B 0,C 180,E1 16788.664,E2 16788.664} C_VEL
LIN {X 0,Y 277.411,Z 1239.803,A -85,B 0,C 180,E1 16794.308,E2 16794.308} C_VEL
LIN {X 0,Y 269.298,Z 1262.632,A -85,B 0,C 180,E1 16801.105,E2 16801.105} C_VEL
LIN {X 0,Y 264.119,Z 1279.319,A -85,B 0,C 180,E1 16808.206,E2 16808.206} C_VEL
LIN {X 0,Y 261.54,Z 1291.299,A -85,B 0,C 180,E1 16815.812,E2 16815.812} C_VEL
LIN {X 0,Y 260.82,Z 1298.085,A -85,B 0,C 180,E1 16823.362,E2 16823.362} C_VEL
LIN {X 0,Y 260.986,Z 1300.07,A -85,B 0,C 180,E1 16830.006,E2 16830.006} C_VEL
LIN {X 0,Y 260.846,Z 1298.089,A -85,B 0,C 180,E1 16836.651,E2 16836.651} C_VEL
LIN {X 0,Y 261.614,Z 1291.304,A -85,B 0,C 180,E1 16844.197,E2 16844.197} C_VEL
LIN {X 0,Y 264.24,Z 1279.331,A -85,B 0,C 180,E1 16851.797,E2 16851.797} C_VEL
LIN {X 0,Y 270.408,Z 1260.327,A -85,B 0,C 180,E1 16859.696,E2 16859.696} C_VEL
LIN {X 0,Y 278.549,Z 1237.833,A -85,B 0,C 180,E1 16866.133,E2 16866.133} C_VEL
LIN {X 0,Y 288.559,Z 1209.717,A -85,B 0,C 180,E1 16871.826,E2 16871.826} C_VEL
LIN {X 0,Y 299.127,Z 1176.492,A -85,B 0,C 180,E1 16876.473,E2 16876.473} C_VEL
LIN {X 0,Y 308.89,Z 1158.063,A -85,B 0,C 180,E1 16879.23,E2 16879.23} C_VEL
LIN {X 0,Y 319.545,Z 1141.181,A -85,B 0,C 180,E1 16881.5,E2 16881.5} C_VEL
LIN {X 0,Y 320.32,Z 1139.779,A -85,B 0,C 180,E1 16881.948,E2 16881.948} C_VEL
LIN {X 0,Y 302.214,Z 1164.354,A -85,B 0,C 180,E1 16886.685,E2 16886.685} C_VEL
LIN {X 0,Y 292.163,Z 1178.405,A -85,B 0,C 180,E1 16890.514,E2 16890.514} C_VEL
LIN {X 0,Y 283.224,Z 1187.805,A -85,B 0,C 180,E1 16892.885,E2 16892.885} C_VEL
LIN {X 0,Y 274.809,Z 1195.641,A -85,B 0,C 180,E1 16895.43,E2 16895.43} C_VEL
LIN {X 0,Y 274.635,Z 1195.781,A -85,B 0,C 180,E1 16895.529,E2 16895.529} C_VEL
LIN {X 0,Y 266.004,Z 1204.746,A -85,B 0,C 180,E1 16901.82,E2 16901.82} C_VEL
LIN {X 0,Y 261.587,Z 1208.322,A -85,B 0,C 180,E1 16906.659,E2 16906.659} C_VEL
LIN {X 0,Y 257.917,Z 1209.232,A -85,B 0,C 180,E1 16913.28,E2 16913.28} C_VEL
LIN {X 0,Y 256.449,Z 1205.611,A -85,B 0,C 180,E1 16919.999,E2 16919.999} C_VEL
LIN {X 0,Y 256.601,Z 1197.213,A -85,B 0,C 180,E1 16926.754,E2 16926.754} C_VEL
LIN {X 0,Y 258.762,Z 1182.149,A -85,B 0,C 180,E1 16933.918,E2 16933.918} C_VEL
LIN {X 0,Y 262.651,Z 1162.096,A -85,B 0,C 180,E1 16940.163,E2 16940.163} C_VEL
LIN {X 0,Y 267.827,Z 1137.758,A -85,B 0,C 180,E1 16945.356,E2 16945.356} C_VEL
LIN {X 0,Y 273.067,Z 1111.166,A -85,B 0,C 180,E1 16949.368,E2 16949.368} C_VEL
LIN {X 0,Y 277.676,Z 1108.202,A -85,B 0,C 180,E1 16950.628,E2 16950.628} C_VEL
LIN {X 0,Y 283.271,Z 1101.324,A -85,B 0,C 180,E1 16951.519,E2 16951.519} C_VEL
LIN {X 0,Y 289.434,Z 1095.771,A -85,B 0,C 180,E1 16952.829,E2 16952.829} C_VEL
LIN {X 0,Y 297.101,Z 1085.428,A -85,B 0,C 180,E1 16953.964,E2 16953.964} C_VEL
LIN {X 0,Y 304.874,Z 1074.478,A -85,B 0,C 180,E1 16955.125,E2 16955.125} C_VEL
LIN {X 0,Y 306.497,Z 1075.691,A -85,B 0,C 180,E1 16955.667,E2 16955.667} C_VEL
LIN {X 0,Y 314.046,Z 1099.689,A -85,B 0,C 180,E1 16959.988,E2 16959.988} C_VEL
LIN {X 0,Y 313.425,Z 1105.514,A -85,B 0,C 180,E1 16960.523,E2 16960.523} C_VEL
LIN {X 0,Y 304.068,Z 1140.064,A -85,B 0,C 180,E1 16963.511,E2 16963.511} C_VEL
LIN {X 0,Y 293.022,Z 1170.954,A -85,B 0,C 180,E1 16967.466,E2 16967.466} C_VEL
LIN {X 0,Y 281.614,Z 1197.741,A -85,B 0,C 180,E1 16972.436,E2 16972.436} C_VEL
LIN {X 0,Y 270.349,Z 1221.467,A -85,B 0,C 180,E1 16978.907,E2 16978.907} C_VEL
LIN {X 0,Y 261.7,Z 1239.258,A -85,B 0,C 180,E1 16986.187,E2 16986.187} C_VEL
LIN {X 0,Y 255.965,Z 1252.245,A -85,B 0,C 180,E1 16994.608,E2 16994.608} C_VEL
LIN {X 0,Y 253.591,Z 1259.13,A -85,B 0,C 180,E1 17003.158,E2 17003.158} C_VEL
LIN {X 0,Y 253.149,Z 1260.831,A -85,B 0,C 180,E1 17009.993,E2 17009.993} C_VEL
LIN {X 0,Y 253.871,Z 1258.135,A -85,B 0,C 180,E1 17018.539,E2 17018.539} C_VEL
LIN {X 0,Y 256.846,Z 1249.998,A -85,B 0,C 180,E1 17027.077,E2 17027.077} C_VEL
LIN {X 0,Y 262.535,Z 1237.414,A -85,B 0,C 180,E1 17034.621,E2 17034.621} C_VEL
LIN {X 0,Y 271.524,Z 1218.823,A -85,B 0,C 180,E1 17041.862,E2 17041.862} C_VEL
LIN {X 0,Y 282.455,Z 1195.672,A -85,B 0,C 180,E1 17047.901,E2 17047.901} C_VEL
LIN {X 0,Y 294.017,Z 1168.237,A -85,B 0,C 180,E1 17052.841,E2 17052.841} C_VEL
LIN {X 0,Y 304.93,Z 1136.828,A -85,B 0,C 180,E1 17056.732,E2 17056.732} C_VEL
LIN {X 0,Y 314.074,Z 1102.398,A -85,B 0,C 180,E1 17059.56,E2 17059.56} C_VEL
LIN {X 0,Y 308.402,Z 1080.958,A -85,B 0,C 180,E1 17063.193,E2 17063.193} C_VEL
LIN {X 0,Y 298.417,Z 1058.082,A -85,B 0,C 180,E1 17067.932,E2 17067.932} C_VEL
LIN {X 0,Y 285.664,Z 1036.517,A -85,B 0,C 180,E1 17073.819,E2 17073.819} C_VEL
LIN {X 0,Y 276.732,Z 1023.624,A -85,B 0,C 180,E1 17078.879,E2 17078.879} C_VEL
LIN {X 0,Y 272.558,Z 1017.515,A -85,B 0,C 180,E1 17081.856,E2 17081.856} C_VEL
LIN {X 0,Y 268.469,Z 1011.414,A -85,B 0,C 180,E1 17085.475,E2 17085.475} C_VEL
LIN {X 0,Y 264.598,Z 1005.494,A -85,B 0,C 180,E1 17090.264,E2 17090.264} C_VEL
LIN {X 0,Y 261.761,Z 1002.923,A -85,B 0,C 180,E1 17096.696,E2 17096.696} C_VEL
LIN {X 0,Y 262.349,Z 1003.494,A -85,B 0,C 180,E1 17104.537,E2 17104.537} C_VEL
LIN {X 0,Y 264.589,Z 1005.439,A -85,B 0,C 180,E1 17108.85,E2 17108.85} C_VEL
LIN {X 0,Y 268.206,Z 1011.27,A -85,B 0,C 180,E1 17113.418,E2 17113.418} C_VEL
LIN {X 0,Y 270,Z 1013.817,A -85,B 0,C 180,E1 17115.135,E2 17115.135} C_VEL
LIN {X 0,Y 275.199,Z 1021.218,A -85,B 0,C 180,E1 17119.208,E2 17119.208} C_VEL
LIN {X 0,Y 283.773,Z 1033.722,A -85,B 0,C 180,E1 17124.343,E2 17124.343} C_VEL
LIN {X 0,Y 286.483,Z 1039.254,A -85,B 0,C 180,E1 17125.801,E2 17125.801} C_VEL
LIN {X 0,Y 301.843,Z 1088.971,A -85,B 0,C 180,E1 17133.683,E2 17133.683} C_VEL
LIN {X 0,Y 307.889,Z 1112.548,A -85,B 0,C 180,E1 17137.141,E2 17137.141} C_VEL
LIN {X 0,Y 300.422,Z 1148.933,A -85,B 0,C 180,E1 17139.613,E2 17139.613} C_VEL
LIN {X 0,Y 290.826,Z 1182.794,A -85,B 0,C 180,E1 17143.129,E2 17143.129} C_VEL
LIN {X 0,Y 280.497,Z 1213.28,A -85,B 0,C 180,E1 17147.748,E2 17147.748} C_VEL
LIN {X 0,Y 270.344,Z 1240.269,A -85,B 0,C 180,E1 17153.563,E2 17153.563} C_VEL
LIN {X 0,Y 262.138,Z 1261.831,A -85,B 0,C 180,E1 17160.166,E2 17160.166} C_VEL
LIN {X 0,Y 256.533,Z 1278.694,A -85,B 0,C 180,E1 17167.527,E2 17167.527} C_VEL
LIN {X 0,Y 253.736,Z 1290.684,A -85,B 0,C 180,E1 17175.366,E2 17175.366} C_VEL
LIN {X 0,Y 252.949,Z 1297.48,A -85,B 0,C 180,E1 17183.154,E2 17183.154} C_VEL
LIN {X 0,Y 253.129,Z 1299.47,A -85,B 0,C 180,E1 17190.007,E2 17190.007} C_VEL
LIN {X 0,Y 252.973,Z 1297.484,A -85,B 0,C 180,E1 17196.859,E2 17196.859} C_VEL
LIN {X 0,Y 253.804,Z 1290.69,A -85,B 0,C 180,E1 17204.644,E2 17204.644} C_VEL
LIN {X 0,Y 256.671,Z 1278.71,A -85,B 0,C 180,E1 17212.474,E2 17212.474} C_VEL
LIN {X 0,Y 263.223,Z 1259.771,A -85,B 0,C 180,E1 17220.564,E2 17220.564} C_VEL
LIN {X 0,Y 272.514,Z 1235.67,A -85,B 0,C 180,E1 17227.534,E2 17227.534} C_VEL
LIN {X 0,Y 283.322,Z 1206.955,A -85,B 0,C 180,E1 17233.303,E2 17233.303} C_VEL
LIN {X 0,Y 293.544,Z 1178.109,A -85,B 0,C 180,E1 17237.498,E2 17237.498} C_VEL
LIN {X 0,Y 310.944,Z 1152.312,A -85,B 0,C 180,E1 17241.629,E2 17241.629} C_VEL
LIN {X 0,Y 311.718,Z 1151.102,A -85,B 0,C 180,E1 17242.054,E2 17242.054} C_VEL
LIN {X 0,Y 292.876,Z 1173.971,A -85,B 0,C 180,E1 17247.249,E2 17247.249} C_VEL
LIN {X 0,Y 278.374,Z 1191.497,A -85,B 0,C 180,E1 17253.435,E2 17253.435} C_VEL
LIN {X 0,Y 274.635,Z 1195.781,A -85,B 0,C 180,E1 17255.529,E2 17255.529} C_VEL
LIN {X 0,Y 266.205,Z 1202.425,A -85,B 0,C 180,E1 17258.479,E2 17258.479} C_VEL
LIN {X 0,Y 259.014,Z 1207.044,A -85,B 0,C 180,E1 17261.246,E2 17261.246} C_VEL
LIN {X 0,Y 258.432,Z 1207.452,A -85,B 0,C 180,E1 17261.702,E2 17261.702} C_VEL
LIN {X 0,Y 251.872,Z 1211.139,A -85,B 0,C 180,E1 17269.645,E2 17269.645} C_VEL
LIN {X 0,Y 249.079,Z 1209.445,A -85,B 0,C 180,E1 17276.526,E2 17276.526} C_VEL
LIN {X 0,Y 248.606,Z 1203.106,A -85,B 0,C 180,E1 17283.479,E2 17283.479} C_VEL
LIN {X 0,Y 249.505,Z 1191.741,A -85,B 0,C 180,E1 17290.452,E2 17290.452} C_VEL
LIN {X 0,Y 252.562,Z 1175.065,A -85,B 0,C 180,E1 17297.038,E2 17297.038} C_VEL
LIN {X 0,Y 257.102,Z 1153.469,A -85,B 0,C 180,E1 17302.881,E2 17302.881} C_VEL
LIN {X 0,Y 262.957,Z 1125.857,A -85,B 0,C 180,E1 17308.022,E2 17308.022} C_VEL
LIN {X 0,Y 267.77,Z 1122.635,A -85,B 0,C 180,E1 17309.543,E2 17309.543} C_VEL
LIN {X 0,Y 273.382,Z 1117.401,A -85,B 0,C 180,E1 17310.7,E2 17310.7} C_VEL
LIN {X 0,Y 280.624,Z 1111.267,A -85,B 0,C 180,E1 17312.189,E2 17312.189} C_VEL
LIN {X 0,Y 284.789,Z 1106.778,A -85,B 0,C 180,E1 17312.894,E2 17312.894} C_VEL
LIN {X 0,Y 293.897,Z 1097.074,A -85,B 0,C 180,E1 17314.385,E2 17314.385} C_VEL
LIN {X 0,Y 303.637,Z 1085.272,A -85,B 0,C 180,E1 17315.816,E2 17315.816} C_VEL
LIN {X 0,Y 308.557,Z 1105.228,A -85,B 0,C 180,E1 17319.354,E2 17319.354} C_VEL
LIN {X 0,Y 298.805,Z 1140.315,A -85,B 0,C 180,E1 17322.379,E2 17322.379} C_VEL
LIN {X 0,Y 287.205,Z 1171.547,A -85,B 0,C 180,E1 17326.392,E2 17326.392} C_VEL
LIN {X 0,Y 275.362,Z 1198.337,A -85,B 0,C 180,E1 17331.429,E2 17331.429} C_VEL
LIN {X 0,Y 263.555,Z 1222.069,A -85,B 0,C 180,E1 17338.012,E2 17338.012} C_VEL
LIN {X 0,Y 254.432,Z 1239.863,A -85,B 0,C 180,E1 17345.462,E2 17345.462} C_VEL
LIN {X 0,Y 248.311,Z 1252.85,A -85,B 0,C 180,E1 17354.122,E2 17354.122} C_VEL
LIN {X 0,Y 245.766,Z 1259.731,A -85,B 0,C 180,E1 17362.939,E2 17362.939} C_VEL
LIN {X 0,Y 245.27,Z 1261.432,A -85,B 0,C 180,E1 17369.993,E2 17369.993} C_VEL
LIN {X 0,Y 246.039,Z 1258.74,A -85,B 0,C 180,E1 17378.813,E2 17378.813} C_VEL
LIN {X 0,Y 249.259,Z 1250.605,A -85,B 0,C 180,E1 17387.613,E2 17387.613} C_VEL
LIN {X 0,Y 255.284,Z 1238.025,A -85,B 0,C 180,E1 17395.369,E2 17395.369} C_VEL
LIN {X 0,Y 264.79,Z 1219.429,A -85,B 0,C 180,E1 17402.772,E2 17402.772} C_VEL
LIN {X 0,Y 276.221,Z 1196.276,A -85,B 0,C 180,E1 17408.915,E2 17408.915} C_VEL
LIN {X 0,Y 288.267,Z 1168.833,A -85,B 0,C 180,E1 17413.91,E2 17413.91} C_VEL
LIN {X 0,Y 299.866,Z 1136.505,A -85,B 0,C 180,E1 17417.918,E2 17417.918} C_VEL
LIN {X 0,Y 308.481,Z 1103.484,A -85,B 0,C 180,E1 17420.741,E2 17420.741} C_VEL
LIN {X 0,Y 300.85,Z 1077.826,A -85,B 0,C 180,E1 17425.576,E2 17425.576} C_VEL
LIN {X 0,Y 290.735,Z 1056.153,A -85,B 0,C 180,E1 17430.672,E2 17430.672} C_VEL
LIN {X 0,Y 279.61,Z 1037.779,A -85,B 0,C 180,E1 17436.444,E2 17436.444} C_VEL
LIN {X 0,Y 270.971,Z 1025.023,A -85,B 0,C 180,E1 17442.271,E2 17442.271} C_VEL
LIN {X 0,Y 266.843,Z 1018.861,A -85,B 0,C 180,E1 17446.072,E2 17446.072} C_VEL
LIN {X 0,Y 263.19,Z 1012.467,A -85,B 0,C 180,E1 17451.01,E2 17451.01} C_VEL
LIN {X 0,Y 260.667,Z 1010.578,A -85,B 0,C 180,E1 17461.659,E2 17461.659} C_VEL
LIN {X 0,Y 263.336,Z 1013.13,A -85,B 0,C 180,E1 17468.447,E2 17468.447} C_VEL
LIN {X 0,Y 267.261,Z 1019.195,A -85,B 0,C 180,E1 17473.466,E2 17473.466} C_VEL
LIN {X 0,Y 273.532,Z 1028.822,A -85,B 0,C 180,E1 17478.807,E2 17478.807} C_VEL
LIN {X 0,Y 282.772,Z 1042.688,A -85,B 0,C 180,E1 17484.435,E2 17484.435} C_VEL
LIN {X 0,Y 296.341,Z 1089.045,A -85,B 0,C 180,E1 17492.105,E2 17492.105} C_VEL
LIN {X 0,Y 302.357,Z 1116.196,A -85,B 0,C 180,E1 17496.156,E2 17496.156} C_VEL
LIN {X 0,Y 294.443,Z 1151.673,A -85,B 0,C 180,E1 17498.702,E2 17498.702} C_VEL
LIN {X 0,Y 284.368,Z 1185.097,A -85,B 0,C 180,E1 17502.31,E2 17502.31} C_VEL
LIN {X 0,Y 272.897,Z 1216.788,A -85,B 0,C 180,E1 17507.368,E2 17507.368} C_VEL
LIN {X 0,Y 262.498,Z 1242.74,A -85,B 0,C 180,E1 17513.355,E2 17513.355} C_VEL
LIN {X 0,Y 253.525,Z 1265.205,A -85,B 0,C 180,E1 17520.796,E2 17520.796} C_VEL
LIN {X 0,Y 248.014,Z 1281.261,A -85,B 0,C 180,E1 17528.595,E2 17528.595} C_VEL
LIN {X 0,Y 245.756,Z 1291.086,A -85,B 0,C 180,E1 17535.789,E2 17535.789} C_VEL
LIN {X 0,Y 245.061,Z 1296.873,A -85,B 0,C 180,E1 17542.932,E2 17542.932} C_VEL
LIN {X 0,Y 245.244,Z 1298.868,A -85,B 0,C 180,E1 17550.007,E2 17550.007} C_VEL
LIN {X 0,Y 245.082,Z 1296.878,A -85,B 0,C 180,E1 17557.081,E2 17557.081} C_VEL
LIN {X 0,Y 245.978,Z 1290.073,A -85,B 0,C 180,E1 17565.121,E2 17565.121} C_VEL
LIN {X 0,Y 249.116,Z 1278.087,A -85,B 0,C 180,E1 17573.195,E2 17573.195} C_VEL
LIN {X 0,Y 256.186,Z 1259.149,A -85,B 0,C 180,E1 17581.498,E2 17581.498} C_VEL
LIN {X 0,Y 266.053,Z 1235.052,A -85,B 0,C 180,E1 17588.611,E2 17588.611} C_VEL
LIN {X 0,Y 277.433,Z 1206.345,A -85,B 0,C 180,E1 17594.461,E2 17594.461} C_VEL
LIN {X 0,Y 286.281,Z 1184.003,A -85,B 0,C 180,E1 17597.949,E2 17597.949} C_VEL
LIN {X 0,Y 302.198,Z 1162.597,A -85,B 0,C 180,E1 17601.775,E2 17601.775} C_VEL
LIN {X 0,Y 302.943,Z 1161.562,A -85,B 0,C 180,E1 17602.178,E2 17602.178} C_VEL
LIN {X 0,Y 283.442,Z 1182.572,A -85,B 0,C 180,E1 17607.834,E2 17607.834} C_VEL
LIN {X 0,Y 267.796,Z 1198.998,A -85,B 0,C 180,E1 17615.001,E2 17615.001} C_VEL
LIN {X 0,Y 258.432,Z 1207.452,A -85,B 0,C 180,E1 17621.702,E2 17621.702} C_VEL
LIN {X 0,Y 251.145,Z 1210.998,A -85,B 0,C 180,E1 17625.205,E2 17625.205} C_VEL
LIN {X 0,Y 244.936,Z 1212.844,A -85,B 0,C 180,E1 17628.421,E2 17628.421} C_VEL
LIN {X 0,Y 244.536,Z 1212.881,A -85,B 0,C 180,E1 17628.923,E2 17628.923} C_VEL
LIN {X 0,Y 241.321,Z 1210.855,A -85,B 0,C 180,E1 17636.414,E2 17636.414} C_VEL
LIN {X 0,Y 240.793,Z 1204.158,A -85,B 0,C 180,E1 17643.592,E2 17643.592} C_VEL
LIN {X 0,Y 241.761,Z 1192.391,A -85,B 0,C 180,E1 17650.791,E2 17650.791} C_VEL
LIN {X 0,Y 245.214,Z 1174.291,A -85,B 0,C 180,E1 17657.919,E2 17657.919} C_VEL
LIN {X 0,Y 250.204,Z 1151.445,A -85,B 0,C 180,E1 17664.021,E2 17664.021} C_VEL
LIN {X 0,Y 253.518,Z 1137.324,A -85,B 0,C 180,E1 17666.901,E2 17666.901} C_VEL
LIN {X 0,Y 256.678,Z 1136.108,A -85,B 0,C 180,E1 17668.053,E2 17668.053} C_VEL
LIN {X 0,Y 262.101,Z 1131.666,A -85,B 0,C 180,E1 17669.297,E2 17669.297} C_VEL
LIN {X 0,Y 268.819,Z 1127.14,A -85,B 0,C 180,E1 17670.971,E2 17670.971} C_VEL
LIN {X 0,Y 281.263,Z 1116.641,A -85,B 0,C 180,E1 17673.359,E2 17673.359} C_VEL
LIN {X 0,Y 295.354,Z 1102.346,A -85,B 0,C 180,E1 17675.513,E2 17675.513} C_VEL
LIN {X 0,Y 300.418,Z 1096.025,A -85,B 0,C 180,E1 17676.133,E2 17676.133} C_VEL
LIN {X 0,Y 302.998,Z 1108.371,A -85,B 0,C 180,E1 17678.372,E2 17678.372} C_VEL
LIN {X 0,Y 293.003,Z 1142.398,A -85,B 0,C 180,E1 17681.402,E2 17681.402} C_VEL
LIN {X 0,Y 281.059,Z 1173.251,A -85,B 0,C 180,E1 17685.456,E2 17685.456} C_VEL
LIN {X 0,Y 268.376,Z 1200.6,A -85,B 0,C 180,E1 17690.751,E2 17690.751} C_VEL
LIN {X 0,Y 256.183,Z 1223.828,A -85,B 0,C 180,E1 17697.478,E2 17697.478} C_VEL
LIN {X 0,Y 247.179,Z 1240.47,A -85,B 0,C 180,E1 17704.693,E2 17704.693} C_VEL
LIN {X 0,Y 240.663,Z 1253.456,A -85,B 0,C 180,E1 17713.603,E2 17713.603} C_VEL
LIN {X 0,Y 237.92,Z 1260.334,A -85,B 0,C 180,E1 17722.705,E2 17722.705} C_VEL
LIN {X 0,Y 237.391,Z 1262.034,A -85,B 0,C 180,E1 17729.993,E2 17729.993} C_VEL
LIN {X 0,Y 238.241,Z 1259.343,A -85,B 0,C 180,E1 17739.104,E2 17739.104} C_VEL
LIN {X 0,Y 241.691,Z 1251.212,A -85,B 0,C 180,E1 17748.184,E2 17748.184} C_VEL
LIN {X 0,Y 248.083,Z 1238.634,A -85,B 0,C 180,E1 17756.161,E2 17756.161} C_VEL
LIN {X 0,Y 258.138,Z 1220.035,A -85,B 0,C 180,E1 17763.728,E2 17763.728} C_VEL
LIN {X 0,Y 270.096,Z 1196.877,A -85,B 0,C 180,E1 17769.972,E2 17769.972} C_VEL
LIN {X 0,Y 282.636,Z 1169.429,A -85,B 0,C 180,E1 17775.019,E2 17775.019} C_VEL
LIN {X 0,Y 294.63,Z 1137.1,A -85,B 0,C 180,E1 17779.057,E2 17779.057} C_VEL
LIN {X 0,Y 302.974,Z 1106.572,A -85,B 0,C 180,E1 17781.724,E2 17781.724} C_VEL
LIN {X 0,Y 295.934,Z 1081.598,A -85,B 0,C 180,E1 17786.651,E2 17786.651} C_VEL
LIN {X 0,Y 286.302,Z 1060.133,A -85,B 0,C 180,E1 17792.005,E2 17792.005} C_VEL
LIN {X 0,Y 276.597,Z 1043.656,A -85,B 0,C 180,E1 17797.551,E2 17797.551} C_VEL
LIN {X 0,Y 269.042,Z 1032.102,A -85,B 0,C 180,E1 17802.981,E2 17802.981} C_VEL
LIN {X 0,Y 265.246,Z 1026.308,A -85,B 0,C 180,E1 17806.676,E2 17806.676} C_VEL
LIN {X 0,Y 261.486,Z 1019.855,A -85,B 0,C 180,E1 17812.245,E2 17812.245} C_VEL
LIN {X 0,Y 259.853,Z 1018.559,A -85,B 0,C 180,E1 17822.497,E2 17822.497} C_VEL
LIN {X 0,Y 262.145,Z 1021.039,A -85,B 0,C 180,E1 17828.149,E2 17828.149} C_VEL
LIN {X 0,Y 267.02,Z 1029.014,A -85,B 0,C 180,E1 17834.308,E2 17834.308} C_VEL
LIN {X 0,Y 272.27,Z 1037.018,A -85,B 0,C 180,E1 17838.688,E2 17838.688} C_VEL
LIN {X 0,Y 280.249,Z 1049.471,A -85,B 0,C 180,E1 17843.716,E2 17843.716} C_VEL
LIN {X 0,Y 291.809,Z 1092.824,A -85,B 0,C 180,E1 17851.03,E2 17851.03} C_VEL
LIN {X 0,Y 297.15,Z 1118.223,A -85,B 0,C 180,E1 17855.056,E2 17855.056} C_VEL
LIN {X 0,Y 288.833,Z 1153.374,A -85,B 0,C 180,E1 17857.661,E2 17857.661} C_VEL
LIN {X 0,Y 277.982,Z 1187.275,A -85,B 0,C 180,E1 17861.434,E2 17861.434} C_VEL
LIN {X 0,Y 266.082,Z 1218.128,A -85,B 0,C 180,E1 17866.566,E2 17866.566} C_VEL
LIN {X 0,Y 255.207,Z 1243.757,A -85,B 0,C 180,E1 17872.715,E2 17872.715} C_VEL
LIN {X 0,Y 245.671,Z 1266.273,A -85,B 0,C 180,E1 17880.575,E2 17880.575} C_VEL
LIN {X 0,Y 239.959,Z 1282.04,A -85,B 0,C 180,E1 17888.803,E2 17888.803} C_VEL
LIN {X 0,Y 237.635,Z 1292.28,A -85,B 0,C 180,E1 17897.165,E2 17897.165} C_VEL
LIN {X 0,Y 237.161,Z 1296.265,A -85,B 0,C 180,E1 17902.696,E2 17902.696} C_VEL
LIN {X 0,Y 237.358,Z 1298.267,A -85,B 0,C 180,E1 17910.007,E2 17910.007} C_VEL
LIN {X 0,Y 237.189,Z 1295.548,A -85,B 0,C 180,E1 17918.651,E2 17918.651} C_VEL
LIN {X 0,Y 238.726,Z 1287.269,A -85,B 0,C 180,E1 17927.481,E2 17927.481} C_VEL
LIN {X 0,Y 243.233,Z 1273.078,A -85,B 0,C 180,E1 17936.272,E2 17936.272} C_VEL
LIN {X 0,Y 251.274,Z 1253.486,A -85,B 0,C 180,E1 17944.273,E2 17944.273} C_VEL
LIN {X 0,Y 262.058,Z 1228.798,A -85,B 0,C 180,E1 17951.104,E2 17951.104} C_VEL
LIN {X 0,Y 273.959,Z 1199.573,A -85,B 0,C 180,E1 17956.676,E2 17956.676} C_VEL
LIN {X 0,Y 278.267,Z 1190.689,A -85,B 0,C 180,E1 17958.226,E2 17958.226} C_VEL
LIN {X 0,Y 292.948,Z 1172.574,A -85,B 0,C 180,E1 17961.821,E2 17961.821} C_VEL
LIN {X 0,Y 293.75,Z 1171.467,A -85,B 0,C 180,E1 17962.41,E2 17962.41} C_VEL
LIN {X 0,Y 273.949,Z 1190.372,A -85,B 0,C 180,E1 17968.447,E2 17968.447} C_VEL
LIN {X 0,Y 258.465,Z 1204.357,A -85,B 0,C 180,E1 17975.878,E2 17975.878} C_VEL
LIN {X 0,Y 249.975,Z 1210.729,A -85,B 0,C 180,E1 17982.432,E2 17982.432} C_VEL
LIN {X 0,Y 244.536,Z 1212.881,A -85,B 0,C 180,E1 17988.923,E2 17988.923} C_VEL
LIN {X 0,Y 240.469,Z 1213.258,A -85,B 0,C 180,E1 17991.869,E2 17991.869} C_VEL
LIN {X 0,Y 233.627,Z 1212.136,A -85,B 0,C 180,E1 17996.35,E2 17996.35} C_VEL
LIN {X 0,Y 233.416,Z 1211.768,A -85,B 0,C 180,E1 17996.878,E2 17996.878} C_VEL
LIN {X 0,Y 232.899,Z 1203.902,A -85,B 0,C 180,E1 18004.645,E2 18004.645} C_VEL
LIN {X 0,Y 234.547,Z 1190.07,A -85,B 0,C 180,E1 18012.54,E2 18012.54} C_VEL
LIN {X 0,Y 238.285,Z 1171.58,A -85,B 0,C 180,E1 18019.417,E2 18019.417} C_VEL
LIN {X 0,Y 243.676,Z 1148.514,A -85,B 0,C 180,E1 18025.441,E2 18025.441} C_VEL
LIN {X 0,Y 249.463,Z 1145.568,A -85,B 0,C 180,E1 18027.433,E2 18027.433} C_VEL
LIN {X 0,Y 267.391,Z 1133.789,A -85,B 0,C 180,E1 18031.911,E2 18031.911} C_VEL
LIN {X 0,Y 282.534,Z 1121.436,A -85,B 0,C 180,E1 18034.601,E2 18034.601} C_VEL
LIN {X 0,Y 297.113,Z 1107.214,A -85,B 0,C 180,E1 18036.669,E2 18036.669} C_VEL
LIN {X 0,Y 297.459,Z 1111.508,A -85,B 0,C 180,E1 18037.372,E2 18037.372} C_VEL
LIN {X 0,Y 287.295,Z 1144.46,A -85,B 0,C 180,E1 18040.383,E2 18040.383} C_VEL
LIN {X 0,Y 274.982,Z 1174.956,A -85,B 0,C 180,E1 18044.478,E2 18044.478} C_VEL
LIN {X 0,Y 261.415,Z 1202.744,A -85,B 0,C 180,E1 18050.035,E2 18050.035} C_VEL
LIN {X 0,Y 248.846,Z 1225.586,A -85,B 0,C 180,E1 18056.914,E2 18056.914} C_VEL
LIN {X 0,Y 239.125,Z 1242.724,A -85,B 0,C 180,E1 18064.78,E2 18064.78} C_VEL
LIN {X 0,Y 233.064,Z 1254.06,A -85,B 0,C 180,E1 18073.053,E2 18073.053} C_VEL
LIN {X 0,Y 230.101,Z 1260.935,A -85,B 0,C 180,E1 18082.456,E2 18082.456} C_VEL
LIN {X 0,Y 229.512,Z 1262.635,A -85,B 0,C 180,E1 18089.993,E2 18089.993} C_VEL
LIN {X 0,Y 230.425,Z 1259.948,A -85,B 0,C 180,E1 18099.416,E2 18099.416} C_VEL
LIN {X 0,Y 234.131,Z 1251.821,A -85,B 0,C 180,E1 18108.793,E2 18108.793} C_VEL
LIN {X 0,Y 240.935,Z 1239.244,A -85,B 0,C 180,E1 18116.999,E2 18116.999} C_VEL
LIN {X 0,Y 251.546,Z 1220.642,A -85,B 0,C 180,E1 18124.736,E2 18124.736} C_VEL
LIN {X 0,Y 264.049,Z 1197.481,A -85,B 0,C 180,E1 18131.081,E2 18131.081} C_VEL
LIN {X 0,Y 277.407,Z 1169.324,A -85,B 0,C 180,E1 18136.287,E2 18136.287} C_VEL
LIN {X 0,Y 289.513,Z 1137.684,A -85,B 0,C 180,E1 18140.24,E2 18140.24} C_VEL
LIN {X 0,Y 297.575,Z 1111.072,A -85,B 0,C 180,E1 18142.52,E2 18142.52} C_VEL
LIN {X 0,Y 292.171,Z 1088.46,A -85,B 0,C 180,E1 18147.08,E2 18147.08} C_VEL
LIN {X 0,Y 283.383,Z 1066.973,A -85,B 0,C 180,E1 18152.554,E2 18152.554} C_VEL
LIN {X 0,Y 274.349,Z 1050.532,A -85,B 0,C 180,E1 18158.208,E2 18158.208} C_VEL
LIN {X 0,Y 266.923,Z 1038.786,A -85,B 0,C 180,E1 18163.917,E2 18163.917} C_VEL
LIN {X 0,Y 263.766,Z 1033.813,A -85,B 0,C 180,E1 18167.193,E2 18167.193} C_VEL
LIN {X 0,Y 260.33,Z 1027.613,A -85,B 0,C 180,E1 18172.588,E2 18172.588} C_VEL
LIN {X 0,Y 258.89,Z 1026.412,A -85,B 0,C 180,E1 18182.506,E2 18182.506} C_VEL
LIN {X 0,Y 260.951,Z 1028.764,A -85,B 0,C 180,E1 18187.8,E2 18187.8} C_VEL
LIN {X 0,Y 265.629,Z 1036.74,A -85,B 0,C 180,E1 18193.967,E2 18193.967} C_VEL
LIN {X 0,Y 270.503,Z 1044.346,A -85,B 0,C 180,E1 18198.183,E2 18198.183} C_VEL
LIN {X 0,Y 277.643,Z 1055.975,A -85,B 0,C 180,E1 18202.906,E2 18202.906} C_VEL
LIN {X 0,Y 287.23,Z 1095.899,A -85,B 0,C 180,E1 18209.831,E2 18209.831} C_VEL
LIN {X 0,Y 291.848,Z 1121.511,A -85,B 0,C 180,E1 18214.006,E2 18214.006} C_VEL
LIN {X 0,Y 282.271,Z 1158.53,A -85,B 0,C 180,E1 18216.912,E2 18216.912} C_VEL
LIN {X 0,Y 271.15,Z 1190.505,A -85,B 0,C 180,E1 18220.696,E2 18220.696} C_VEL
LIN {X 0,Y 258.88,Z 1220.454,A -85,B 0,C 180,E1 18225.921,E2 18225.921} C_VEL
LIN {X 0,Y 246.882,Z 1247.096,A -85,B 0,C 180,E1 18232.758,E2 18232.758} C_VEL
LIN {X 0,Y 237.657,Z 1267.67,A -85,B 0,C 180,E1 18240.529,E2 18240.529} C_VEL
LIN {X 0,Y 231.933,Z 1282.832,A -85,B 0,C 180,E1 18249.039,E2 18249.039} C_VEL
LIN {X 0,Y 229.792,Z 1291.665,A -85,B 0,C 180,E1 18256.719,E2 18256.719} C_VEL
LIN {X 0,Y 229.268,Z 1295.657,A -85,B 0,C 180,E1 18262.443,E2 18262.443} C_VEL
LIN {X 0,Y 229.472,Z 1297.665,A -85,B 0,C 180,E1 18270.007,E2 18270.007} C_VEL
LIN {X 0,Y 229.287,Z 1295.663,A -85,B 0,C 180,E1 18277.571,E2 18277.571} C_VEL
LIN {X 0,Y 230.428,Z 1288.843,A -85,B 0,C 180,E1 18286.168,E2 18286.168} C_VEL
LIN {X 0,Y 234.501,Z 1276.068,A -85,B 0,C 180,E1 18295.228,E2 18295.228} C_VEL
LIN {X 0,Y 242.366,Z 1257.639,A -85,B 0,C 180,E1 18303.635,E2 18303.635} C_VEL
LIN {X 0,Y 253.362,Z 1233.81,A -85,B 0,C 180,E1 18310.941,E2 18310.941} C_VEL
LIN {X 0,Y 265.994,Z 1205.013,A -85,B 0,C 180,E1 18316.96,E2 18316.96} C_VEL
LIN {X 0,Y 269.932,Z 1197.26,A -85,B 0,C 180,E1 18318.403,E2 18318.403} C_VEL
LIN {X 0,Y 283.98,Z 1181.294,A -85,B 0,C 180,E1 18321.966,E2 18321.966} C_VEL
LIN {X 0,Y 284.925,Z 1180.14,A -85,B 0,C 180,E1 18322.543,E2 18322.543} C_VEL
LIN {X 0,Y 264.438,Z 1197.353,A -85,B 0,C 180,E1 18329.098,E2 18329.098} C_VEL
LIN {X 0,Y 249.247,Z 1209.023,A -85,B 0,C 180,E1 18336.826,E2 18336.826} C_VEL
LIN {X 0,Y 239.362,Z 1214.344,A -85,B 0,C 180,E1 18345.394,E2 18345.394} C_VEL
LIN {X 0,Y 234.9,Z 1213.969,A -85,B 0,C 180,E1 18352.618,E2 18352.618} C_VEL
LIN {X 0,Y 233.416,Z 1211.768,A -85,B 0,C 180,E1 18356.878,E2 18356.878} C_VEL
LIN {X 0,Y 231.829,Z 1210.356,A -85,B 0,C 180,E1 18358.97,E2 18358.97} C_VEL
LIN {X 0,Y 225.168,Z 1204.974,A -85,B 0,C 180,E1 18364.679,E2 18364.679} C_VEL
LIN {X 0,Y 225.101,Z 1204.243,A -85,B 0,C 180,E1 18365.209,E2 18365.209} C_VEL
LIN {X 0,Y 227.059,Z 1189.447,A -85,B 0,C 180,E1 18373.449,E2 18373.449} C_VEL
LIN {X 0,Y 231.135,Z 1170.158,A -85,B 0,C 180,E1 18380.542,E2 18380.542} C_VEL
LIN {X 0,Y 233.899,Z 1158.687,A -85,B 0,C 180,E1 18383.778,E2 18383.778} C_VEL
LIN {X 0,Y 237.479,Z 1157.424,A -85,B 0,C 180,E1 18385.397,E2 18385.397} C_VEL
LIN {X 0,Y 256.875,Z 1146.02,A -85,B 0,C 180,E1 18390.929,E2 18390.929} C_VEL
LIN {X 0,Y 269.192,Z 1137.632,A -85,B 0,C 180,E1 18393.481,E2 18393.481} C_VEL
LIN {X 0,Y 283.527,Z 1126.378,A -85,B 0,C 180,E1 18395.832,E2 18395.832} C_VEL
LIN {X 0,Y 289.968,Z 1120.917,A -85,B 0,C 180,E1 18396.746,E2 18396.746} C_VEL
LIN {X 0,Y 278.965,Z 1153.617,A -85,B 0,C 180,E1 18400.165,E2 18400.165} C_VEL
LIN {X 0,Y 266.001,Z 1182.832,A -85,B 0,C 180,E1 18404.537,E2 18404.537} C_VEL
LIN {X 0,Y 252.057,Z 1209.317,A -85,B 0,C 180,E1 18410.434,E2 18410.434} C_VEL
LIN {X 0,Y 239.538,Z 1230.546,A -85,B 0,C 180,E1 18417.615,E2 18417.615} C_VEL
LIN {X 0,Y 230.17,Z 1246.257,A -85,B 0,C 180,E1 18425.802,E2 18425.802} C_VEL
LIN {X 0,Y 224.575,Z 1256.475,A -85,B 0,C 180,E1 18434.4,E2 18434.4} C_VEL
LIN {X 0,Y 222.274,Z 1261.538,A -85,B 0,C 180,E1 18442.189,E2 18442.189} C_VEL
LIN {X 0,Y 221.638,Z 1263.236,A -85,B 0,C 180,E1 18449.992,E2 18449.992} C_VEL
LIN {X 0,Y 222.567,Z 1260.698,A -85,B 0,C 180,E1 18459.498,E2 18459.498} C_VEL
LIN {X 0,Y 226.627,Z 1252.427,A -85,B 0,C 180,E1 18469.439,E2 18469.439} C_VEL
LIN {X 0,Y 233.859,Z 1239.852,A -85,B 0,C 180,E1 18477.886,E2 18477.886} C_VEL
LIN {X 0,Y 245.032,Z 1221.249,A -85,B 0,C 180,E1 18485.799,E2 18485.799} C_VEL
LIN {X 0,Y 258.106,Z 1198.084,A -85,B 0,C 180,E1 18492.241,E2 18492.241} C_VEL
LIN {X 0,Y 271.461,Z 1171.054,A -85,B 0,C 180,E1 18497.318,E2 18497.318} C_VEL
LIN {X 0,Y 283.978,Z 1139.925,A -85,B 0,C 180,E1 18501.296,E2 18501.296} C_VEL
LIN {X 0,Y 292.143,Z 1112.756,A -85,B 0,C 180,E1 18503.773,E2 18503.773} C_VEL
LIN {X 0,Y 286.322,Z 1088.885,A -85,B 0,C 180,E1 18508.978,E2 18508.978} C_VEL
LIN {X 0,Y 277.411,Z 1067.553,A -85,B 0,C 180,E1 18515.068,E2 18515.068} C_VEL
LIN {X 0,Y 269.368,Z 1052.828,A -85,B 0,C 180,E1 18520.892,E2 18520.892} C_VEL
LIN {X 0,Y 263.003,Z 1041.891,A -85,B 0,C 180,E1 18526.944,E2 18526.944} C_VEL
LIN {X 0,Y 259.187,Z 1035.339,A -85,B 0,C 180,E1 18532.935,E2 18532.935} C_VEL
LIN {X 0,Y 257.927,Z 1034.266,A -85,B 0,C 180,E1 18542.515,E2 18542.515} C_VEL
LIN {X 0,Y 259.768,Z 1036.483,A -85,B 0,C 180,E1 18547.448,E2 18547.448} C_VEL
LIN {X 0,Y 264.158,Z 1044.263,A -85,B 0,C 180,E1 18553.523,E2 18553.523} C_VEL
LIN {X 0,Y 270.709,Z 1054.517,A -85,B 0,C 180,E1 18559.116,E2 18559.116} C_VEL
LIN {X 0,Y 275.31,Z 1063.444,A -85,B 0,C 180,E1 18562.257,E2 18562.257} C_VEL
LIN {X 0,Y 283.592,Z 1103.542,A -85,B 0,C 180,E1 18569.391,E2 18569.391} C_VEL
LIN {X 0,Y 286.611,Z 1124.731,A -85,B 0,C 180,E1 18572.916,E2 18572.916} C_VEL
LIN {X 0,Y 276.733,Z 1160.188,A -85,B 0,C 180,E1 18575.8,E2 18575.8} C_VEL
LIN {X 0,Y 264.902,Z 1192.45,A -85,B 0,C 180,E1 18579.741,E2 18579.741} C_VEL
LIN {X 0,Y 252.151,Z 1221.85,A -85,B 0,C 180,E1 18585.053,E2 18585.053} C_VEL
LIN {X 0,Y 239.755,Z 1247.7,A -85,B 0,C 180,E1 18591.97,E2 18591.97} C_VEL
LIN {X 0,Y 230.085,Z 1268.055,A -85,B 0,C 180,E1 18600.002,E2 18600.002} C_VEL
LIN {X 0,Y 223.872,Z 1283.586,A -85,B 0,C 180,E1 18609.283,E2 18609.283} C_VEL
LIN {X 0,Y 221.687,Z 1292.675,A -85,B 0,C 180,E1 18618.224,E2 18618.224} C_VEL
LIN {X 0,Y 221.341,Z 1296.511,A -85,B 0,C 180,E1 18626.098,E2 18626.098} C_VEL
LIN {X 0,Y 221.595,Z 1297.064,A -85,B 0,C 180,E1 18630.008,E2 18630.008} C_VEL
LIN {X 0,Y 221.422,Z 1295.058,A -85,B 0,C 180,E1 18637.842,E2 18637.842} C_VEL
LIN {X 0,Y 222.397,Z 1289.247,A -85,B 0,C 180,E1 18645.756,E2 18645.756} C_VEL
LIN {X 0,Y 226.451,Z 1276.981,A -85,B 0,C 180,E1 18655.176,E2 18655.176} C_VEL
LIN {X 0,Y 234.269,Z 1259.7,A -85,B 0,C 180,E1 18663.684,E2 18663.684} C_VEL
LIN {X 0,Y 245.674,Z 1236.465,A -85,B 0,C 180,E1 18671.333,E2 18671.333} C_VEL
LIN {X 0,Y 257.968,Z 1210.045,A -85,B 0,C 180,E1 18677.247,E2 18677.247} C_VEL
LIN {X 0,Y 262.655,Z 1202.09,A -85,B 0,C 180,E1 18678.955,E2 18678.955} C_VEL
LIN {X 0,Y 275.54,Z 1188.7,A -85,B 0,C 180,E1 18682.258,E2 18682.258} C_VEL
LIN {X 0,Y 275.171,Z 1188.7,A -85,B 0,C 180,E1 18682.9,E2 18682.9} C_VEL
LIN {X 0,Y 253.611,Z 1204.482,A -85,B 0,C 180,E1 18690.273,E2 18690.273} C_VEL
LIN {X 0,Y 239.885,Z 1213.144,A -85,B 0,C 180,E1 18697.826,E2 18697.826} C_VEL
LIN {X 0,Y 231.982,Z 1216.323,A -85,B 0,C 180,E1 18704.918,E2 18704.918} C_VEL
LIN {X 0,Y 227.208,Z 1215.495,A -85,B 0,C 180,E1 18712.366,E2 18712.366} C_VEL
LIN {X 0,Y 225.143,Z 1209.422,A -85,B 0,C 180,E1 18720.959,E2 18720.959} C_VEL
LIN {X 0,Y 225.101,Z 1204.243,A -85,B 0,C 180,E1 18725.209,E2 18725.209} C_VEL
LIN {X 0,Y 221.782,Z 1198.29,A -85,B 0,C 180,E1 18729.341,E2 18729.341} C_VEL
LIN {X 0,Y 219.162,Z 1190.897,A -85,B 0,C 180,E1 18733.442,E2 18733.442} C_VEL
LIN {X 0,Y 223.326,Z 1171.58,A -85,B 0,C 180,E1 18740.776,E2 18740.776} C_VEL
LIN {X 0,Y 224.58,Z 1168.156,A -85,B 0,C 180,E1 18742.205,E2 18742.205} C_VEL
LIN {X 0,Y 242.343,Z 1159.335,A -85,B 0,C 180,E1 18748.75,E2 18748.75} C_VEL
LIN {X 0,Y 264.025,Z 1146.692,A -85,B 0,C 180,E1 18753.863,E2 18753.863} C_VEL
LIN {X 0,Y 281.229,Z 1134.244,A -85,B 0,C 180,E1 18756.648,E2 18756.648} C_VEL
LIN {X 0,Y 268.742,Z 1166.19,A -85,B 0,C 180,E1 18760.49,E2 18760.49} C_VEL
LIN {X 0,Y 254.716,Z 1194.465,A -85,B 0,C 180,E1 18765.463,E2 18765.463} C_VEL
LIN {X 0,Y 240.898,Z 1218.288,A -85,B 0,C 180,E1 18771.777,E2 18771.777} C_VEL
LIN {X 0,Y 228.983,Z 1237.196,A -85,B 0,C 180,E1 18779.355,E2 18779.355} C_VEL
LIN {X 0,Y 220.052,Z 1251.578,A -85,B 0,C 180,E1 18788.452,E2 18788.452} C_VEL
LIN {X 0,Y 215.367,Z 1260.092,A -85,B 0,C 180,E1 18797.858,E2 18797.858} C_VEL
LIN {X 0,Y 213.851,Z 1263.394,A -85,B 0,C 180,E1 18805.946,E2 18805.946} C_VEL
LIN {X 0,Y 213.905,Z 1263.363,A -85,B 0,C 180,E1 18814.038,E2 18814.038} C_VEL
LIN {X 0,Y 215.355,Z 1260.031,A -85,B 0,C 180,E1 18822.127,E2 18822.127} C_VEL
LIN {X 0,Y 220.134,Z 1251.392,A -85,B 0,C 180,E1 18831.566,E2 18831.566} C_VEL
LIN {X 0,Y 229.136,Z 1236.868,A -85,B 0,C 180,E1 18840.682,E2 18840.682} C_VEL
LIN {X 0,Y 241.729,Z 1216.753,A -85,B 0,C 180,E1 18848.62,E2 18848.62} C_VEL
LIN {X 0,Y 256.062,Z 1191.67,A -85,B 0,C 180,E1 18854.998,E2 18854.998} C_VEL
LIN {X 0,Y 269.985,Z 1163.121,A -85,B 0,C 180,E1 18859.832,E2 18859.832} C_VEL
LIN {X 0,Y 282.592,Z 1130.646,A -85,B 0,C 180,E1 18863.518,E2 18863.518} C_VEL
LIN {X 0,Y 286.83,Z 1115.912,A -85,B 0,C 180,E1 18864.839,E2 18864.839} C_VEL
LIN {X 0,Y 281.449,Z 1092.408,A -85,B 0,C 180,E1 18870.269,E2 18870.269} C_VEL
LIN {X 0,Y 273.169,Z 1071.188,A -85,B 0,C 180,E1 18876.716,E2 18876.716} C_VEL
LIN {X 0,Y 264.862,Z 1055.198,A -85,B 0,C 180,E1 18883.77,E2 18883.77} C_VEL
LIN {X 0,Y 260.66,Z 1048.495,A -85,B 0,C 180,E1 18888.527,E2 18888.527} C_VEL
LIN {X 0,Y 258.053,Z 1043.073,A -85,B 0,C 180,E1 18893.285,E2 18893.285} C_VEL
LIN {X 0,Y 256.967,Z 1042.101,A -85,B 0,C 180,E1 18902.525,E2 18902.525} C_VEL
LIN {X 0,Y 258.627,Z 1044.34,A -85,B 0,C 180,E1 18907.176,E2 18907.176} C_VEL
LIN {X 0,Y 262.888,Z 1052.083,A -85,B 0,C 180,E1 18913.274,E2 18913.274} C_VEL
LIN {X 0,Y 269.032,Z 1062.175,A -85,B 0,C 180,E1 18918.709,E2 18918.709} C_VEL
LIN {X 0,Y 272.501,Z 1069.336,A -85,B 0,C 180,E1 18921.309,E2 18921.309} C_VEL
LIN {X 0,Y 279.158,Z 1107.383,A -85,B 0,C 180,E1 18928.286,E2 18928.286} C_VEL
LIN {X 0,Y 281.427,Z 1127.658,A -85,B 0,C 180,E1 18931.781,E2 18931.781} C_VEL
LIN {X 0,Y 270.913,Z 1163.019,A -85,B 0,C 180,E1 18934.764,E2 18934.764} C_VEL
LIN {X 0,Y 258.203,Z 1195.596,A -85,B 0,C 180,E1 18938.928,E2 18938.928} C_VEL
LIN {X 0,Y 244.652,Z 1224.723,A -85,B 0,C 180,E1 18944.515,E2 18944.515} C_VEL
LIN {X 0,Y 231.798,Z 1250.001,A -85,B 0,C 180,E1 18951.703,E2 18951.703} C_VEL
LIN {X 0,Y 221.595,Z 1270.316,A -85,B 0,C 180,E1 18960.423,E2 18960.423} C_VEL
LIN {X 0,Y 215.825,Z 1284.178,A -85,B 0,C 180,E1 18969.545,E2 18969.545} C_VEL
LIN {X 0,Y 213.844,Z 1292.063,A -85,B 0,C 180,E1 18977.786,E2 18977.786} C_VEL
LIN {X 0,Y 213.44,Z 1295.906,A -85,B 0,C 180,E1 18985.954,E2 18985.954} C_VEL
LIN {X 0,Y 213.707,Z 1296.462,A -85,B 0,C 180,E1 18990.008,E2 18990.008} C_VEL
LIN {X 0,Y 213.538,Z 1294.335,A -85,B 0,C 180,E1 18998.387,E2 18998.387} C_VEL
LIN {X 0,Y 215.085,Z 1287.13,A -85,B 0,C 180,E1 19007.853,E2 19007.853} C_VEL
LIN {X 0,Y 220.112,Z 1274.122,A -85,B 0,C 180,E1 19017.481,E2 19017.481} C_VEL
LIN {X 0,Y 229.315,Z 1255.338,A -85,B 0,C 180,E1 19026.327,E2 19026.327} C_VEL
LIN {X 0,Y 241.853,Z 1231.252,A -85,B 0,C 180,E1 19033.849,E2 19033.849} C_VEL
LIN {X 0,Y 253.27,Z 1208.856,A -85,B 0,C 180,E1 19038.866,E2 19038.866} C_VEL
LIN {X 0,Y 266.489,Z 1196.029,A -85,B 0,C 180,E1 19042.457,E2 19042.457} C_VEL
LIN {X 0,Y 265.232,Z 1196.559,A -85,B 0,C 180,E1 19043.316,E2 19043.316} C_VEL
LIN {X 0,Y 245.067,Z 1209.312,A -85,B 0,C 180,E1 19050.489,E2 19050.489} C_VEL
LIN {X 0,Y 233.002,Z 1215.709,A -85,B 0,C 180,E1 19057.134,E2 19057.134} C_VEL
LIN {X 0,Y 224.626,Z 1218.325,A -85,B 0,C 180,E1 19064.412,E2 19064.412} C_VEL
LIN {X 0,Y 218.682,Z 1216.044,A -85,B 0,C 180,E1 19074.058,E2 19074.058} C_VEL
LIN {X 0,Y 217.296,Z 1208.18,A -85,B 0,C 180,E1 19082.985,E2 19082.985} C_VEL
LIN {X 0,Y 218.237,Z 1195.928,A -85,B 0,C 180,E1 19090.96,E2 19090.96} C_VEL
LIN {X 0,Y 219.162,Z 1190.897,A -85,B 0,C 180,E1 19093.442,E2 19093.442} C_VEL
LIN {X 0,Y 216.428,Z 1185.504,A -85,B 0,C 180,E1 19096.116,E2 19096.116} C_VEL
LIN {X 0,Y 213.985,Z 1179.505,A -85,B 0,C 180,E1 19098.768,E2 19098.768} C_VEL
LIN {X 0,Y 214.915,Z 1176.909,A -85,B 0,C 180,E1 19100.015,E2 19100.015} C_VEL
LIN {X 0,Y 231.178,Z 1169.641,A -85,B 0,C 180,E1 19107.187,E2 19107.187} C_VEL
LIN {X 0,Y 253.911,Z 1157.734,A -85,B 0,C 180,E1 19113.215,E2 19113.215} C_VEL
LIN {X 0,Y 271.693,Z 1146.521,A -85,B 0,C 180,E1 19116.395,E2 19116.395} C_VEL
LIN {X 0,Y 271.588,Z 1148.615,A -85,B 0,C 180,E1 19116.854,E2 19116.854} C_VEL
LIN {X 0,Y 257.277,Z 1179.943,A -85,B 0,C 180,E1 19121.268,E2 19121.268} C_VEL
LIN {X 0,Y 242.666,Z 1206.084,A -85,B 0,C 180,E1 19126.83,E2 19126.83} C_VEL
LIN {X 0,Y 228.45,Z 1228.549,A -85,B 0,C 180,E1 19134.1,E2 19134.1} C_VEL
LIN {X 0,Y 216.678,Z 1246.012,A -85,B 0,C 180,E1 19143.075,E2 19143.075} C_VEL
LIN {X 0,Y 210.356,Z 1255.876,A -85,B 0,C 180,E1 19151.158,E2 19151.158} C_VEL
LIN {X 0,Y 206.63,Z 1262.743,A -85,B 0,C 180,E1 19161.593,E2 19161.593} C_VEL
LIN {X 0,Y 205.887,Z 1264.438,A -85,B 0,C 180,E1 19169.992,E2 19169.992} C_VEL
LIN {X 0,Y 206.634,Z 1262.698,A -85,B 0,C 180,E1 19178.391,E2 19178.391} C_VEL
LIN {X 0,Y 210.409,Z 1255.781,A -85,B 0,C 180,E1 19188.82,E2 19188.82} C_VEL
LIN {X 0,Y 218.774,Z 1242.723,A -85,B 0,C 180,E1 19198.863,E2 19198.863} C_VEL
LIN {X 0,Y 231.409,Z 1223.837,A -85,B 0,C 180,E1 19207.608,E2 19207.608} C_VEL
LIN {X 0,Y 246.1,Z 1200.114,A -85,B 0,C 180,E1 19214.533,E2 19214.533} C_VEL
LIN {X 0,Y 260.612,Z 1173.01,A -85,B 0,C 180,E1 19219.752,E2 19219.752} C_VEL
LIN {X 0,Y 274.381,Z 1141.104,A -85,B 0,C 180,E1 19223.87,E2 19223.87} C_VEL
LIN {X 0,Y 281.578,Z 1119.091,A -85,B 0,C 180,E1 19225.954,E2 19225.954} C_VEL
LIN {X 0,Y 277.196,Z 1097.688,A -85,B 0,C 180,E1 19231.119,E2 19231.119} C_VEL
LIN {X 0,Y 269.988,Z 1077.444,A -85,B 0,C 180,E1 19237.513,E2 19237.513} C_VEL
LIN {X 0,Y 262.813,Z 1062.257,A -85,B 0,C 180,E1 19244.495,E2 19244.495} C_VEL
LIN {X 0,Y 259.066,Z 1055.759,A -85,B 0,C 180,E1 19249.195,E2 19249.195} C_VEL
LIN {X 0,Y 256.909,Z 1050.803,A -85,B 0,C 180,E1 19253.678,E2 19253.678} C_VEL
LIN {X 0,Y 256.003,Z 1049.957,A -85,B 0,C 180,E1 19262.534,E2 19262.534} C_VEL
LIN {X 0,Y 257.487,Z 1052.108,A -85,B 0,C 180,E1 19266.872,E2 19266.872} C_VEL
LIN {X 0,Y 261.61,Z 1059.943,A -85,B 0,C 180,E1 19273.022,E2 19273.022} C_VEL
LIN {X 0,Y 267.419,Z 1070.273,A -85,B 0,C 180,E1 19278.506,E2 19278.506} C_VEL
LIN {X 0,Y 269.806,Z 1075.788,A -85,B 0,C 180,E1 19280.46,E2 19280.46} C_VEL
LIN {X 0,Y 275.168,Z 1114.58,A -85,B 0,C 180,E1 19287.785,E2 19287.785} C_VEL
LIN {X 0,Y 276.473,Z 1130.117,A -85,B 0,C 180,E1 19290.57,E2 19290.57} C_VEL
LIN {X 0,Y 265.163,Z 1165.751,A -85,B 0,C 180,E1 19293.674,E2 19293.674} C_VEL
LIN {X 0,Y 251.867,Z 1197.73,A -85,B 0,C 180,E1 19297.939,E2 19297.939} C_VEL
LIN {X 0,Y 238.495,Z 1225.001,A -85,B 0,C 180,E1 19303.323,E2 19303.323} C_VEL
LIN {X 0,Y 225.107,Z 1249.925,A -85,B 0,C 180,E1 19310.596,E2 19310.596} C_VEL
LIN {X 0,Y 214.488,Z 1269.719,A -85,B 0,C 180,E1 19319.358,E2 19319.358} C_VEL
LIN {X 0,Y 208.215,Z 1283.557,A -85,B 0,C 180,E1 19328.762,E2 19328.762} C_VEL
LIN {X 0,Y 205.99,Z 1291.449,A -85,B 0,C 180,E1 19337.312,E2 19337.312} C_VEL
LIN {X 0,Y 205.538,Z 1295.302,A -85,B 0,C 180,E1 19345.798,E2 19345.798} C_VEL
LIN {X 0,Y 205.83,Z 1295.86,A -85,B 0,C 180,E1 19350.008,E2 19350.008} C_VEL
LIN {X 0,Y 205.663,Z 1293.844,A -85,B 0,C 180,E1 19358.447,E2 19358.447} C_VEL
LIN {X 0,Y 206.889,Z 1288.016,A -85,B 0,C 180,E1 19366.972,E2 19366.972} C_VEL
LIN {X 0,Y 211.401,Z 1276.501,A -85,B 0,C 180,E1 19376.564,E2 19376.564} C_VEL
LIN {X 0,Y 220.603,Z 1258.633,A -85,B 0,C 180,E1 19385.985,E2 19385.985} C_VEL
LIN {X 0,Y 233.534,Z 1235.223,A -85,B 0,C 180,E1 19394.009,E2 19394.009} C_VEL
LIN {X 0,Y 245.335,Z 1213.537,A -85,B 0,C 180,E1 19399.278,E2 19399.278} C_VEL
LIN {X 0,Y 257.267,Z 1202.79,A -85,B 0,C 180,E1 19402.638,E2 19402.638} C_VEL
LIN {X 0,Y 256.966,Z 1202.689,A -85,B 0,C 180,E1 19403.226,E2 19403.226} C_VEL
LIN {X 0,Y 235.316,Z 1214.311,A -85,B 0,C 180,E1 19411.253,E2 19411.253} C_VEL
LIN {X 0,Y 221.309,Z 1219.694,A -85,B 0,C 180,E1 19420.067,E2 19420.067} C_VEL
LIN {X 0,Y 214.083,Z 1219.901,A -85,B 0,C 180,E1 19427.792,E2 19427.792} C_VEL
LIN {X 0,Y 210.244,Z 1216.063,A -85,B 0,C 180,E1 19435.884,E2 19435.884} C_VEL
LIN {X 0,Y 209.479,Z 1207.783,A -85,B 0,C 180,E1 19444.13,E2 19444.13} C_VEL
LIN {X 0,Y 211.031,Z 1193.332,A -85,B 0,C 180,E1 19452.911,E2 19452.911} C_VEL
LIN {X 0,Y 213.985,Z 1179.505,A -85,B 0,C 180,E1 19458.768,E2 19458.768} C_VEL
LIN {X 0,Y 215.23,Z 1178.044,A -85,B 0,C 180,E1 19461.022,E2 19461.022} C_VEL
LIN {X 0,Y 218.204,Z 1179.83,A -85,B 0,C 180,E1 19464.557,E2 19464.557} C_VEL
LIN {X 0,Y 218.934,Z 1179.577,A -85,B 0,C 180,E1 19464.9,E2 19464.9} C_VEL
LIN {X 0,Y 241.668,Z 1169.035,A -85,B 0,C 180,E1 19472.054,E2 19472.054} C_VEL
LIN {X 0,Y 261.649,Z 1158.25,A -85,B 0,C 180,E1 19476.142,E2 19476.142} C_VEL
LIN {X 0,Y 263.091,Z 1158.07,A -85,B 0,C 180,E1 19476.57,E2 19476.57} C_VEL
LIN {X 0,Y 248.252,Z 1187.651,A -85,B 0,C 180,E1 19481.205,E2 19481.205} C_VEL
LIN {X 0,Y 233.121,Z 1212.661,A -85,B 0,C 180,E1 19487.171,E2 19487.171} C_VEL
LIN {X 0,Y 219.002,Z 1233.396,A -85,B 0,C 180,E1 19494.745,E2 19494.745} C_VEL
LIN {X 0,Y 207.595,Z 1249.512,A -85,B 0,C 180,E1 19504.132,E2 19504.132} C_VEL
LIN {X 0,Y 200.705,Z 1259.88,A -85,B 0,C 180,E1 19514.734,E2 19514.734} C_VEL
LIN {X 0,Y 198.823,Z 1263.345,A -85,B 0,C 180,E1 19521.26,E2 19521.26} C_VEL
LIN {X 0,Y 198.008,Z 1265.039,A -85,B 0,C 180,E1 19529.992,E2 19529.992} C_VEL
LIN {X 0,Y 198.979,Z 1262.963,A -85,B 0,C 180,E1 19539.658,E2 19539.658} C_VEL
LIN {X 0,Y 203.546,Z 1255.334,A -85,B 0,C 180,E1 19550.611,E2 19550.611} C_VEL
LIN {X 0,Y 212.744,Z 1242.063,A -85,B 0,C 180,E1 19560.662,E2 19560.662} C_VEL
LIN {X 0,Y 226.237,Z 1222.815,A -85,B 0,C 180,E1 19569.435,E2 19569.435} C_VEL
LIN {X 0,Y 241.412,Z 1199.193,A -85,B 0,C 180,E1 19576.217,E2 19576.217} C_VEL
LIN {X 0,Y 256.628,Z 1171.516,A -85,B 0,C 180,E1 19581.444,E2 19581.444} C_VEL
LIN {X 0,Y 270.413,Z 1140.039,A -85,B 0,C 180,E1 19585.389,E2 19585.389} C_VEL
LIN {X 0,Y 276.404,Z 1122.12,A -85,B 0,C 180,E1 19587.146,E2 19587.146} C_VEL
LIN {X 0,Y 272.735,Z 1101.959,A -85,B 0,C 180,E1 19592.274,E2 19592.274} C_VEL
LIN {X 0,Y 266.406,Z 1082.754,A -85,B 0,C 180,E1 19598.725,E2 19598.725} C_VEL
LIN {X 0,Y 260.368,Z 1068.942,A -85,B 0,C 180,E1 19605.42,E2 19605.42} C_VEL
LIN {X 0,Y 257.535,Z 1063.245,A -85,B 0,C 180,E1 19609.664,E2 19609.664} C_VEL
LIN {X 0,Y 255.641,Z 1058.509,A -85,B 0,C 180,E1 19614.072,E2 19614.072} C_VEL
LIN {X 0,Y 255.008,Z 1057.79,A -85,B 0,C 180,E1 19622.544,E2 19622.544} C_VEL
LIN {X 0,Y 256.334,Z 1059.97,A -85,B 0,C 180,E1 19626.656,E2 19626.656} C_VEL
LIN {X 0,Y 260.064,Z 1067.553,A -85,B 0,C 180,E1 19632.674,E2 19632.674} C_VEL
LIN {X 0,Y 265.832,Z 1078.714,A -85,B 0,C 180,E1 19638.513,E2 19638.513} C_VEL
LIN {X 0,Y 267.153,Z 1083.742,A -85,B 0,C 180,E1 19639.918,E2 19639.918} C_VEL
LIN {X 0,Y 271.121,Z 1123.33,A -85,B 0,C 180,E1 19647.592,E2 19647.592} C_VEL
LIN {X 0,Y 271.485,Z 1133.153,A -85,B 0,C 180,E1 19649.359,E2 19649.359} C_VEL
LIN {X 0,Y 259.523,Z 1168.238,A -85,B 0,C 180,E1 19652.539,E2 19652.539} C_VEL
LIN {X 0,Y 246.331,Z 1198.362,A -85,B 0,C 180,E1 19656.65,E2 19656.65} C_VEL
LIN {X 0,Y 231.978,Z 1226.16,A -85,B 0,C 180,E1 19662.283,E2 19662.283} C_VEL
LIN {X 0,Y 218.028,Z 1250.594,A -85,B 0,C 180,E1 19669.707,E2 19669.707} C_VEL
LIN {X 0,Y 207.362,Z 1269.207,A -85,B 0,C 180,E1 19678.264,E2 19678.264} C_VEL
LIN {X 0,Y 200.641,Z 1282.935,A -85,B 0,C 180,E1 19687.919,E2 19687.919} C_VEL
LIN {X 0,Y 198.168,Z 1290.836,A -85,B 0,C 180,E1 19696.803,E2 19696.803} C_VEL
LIN {X 0,Y 197.636,Z 1294.697,A -85,B 0,C 180,E1 19705.629,E2 19705.629} C_VEL
LIN {X 0,Y 197.94,Z 1295.258,A -85,B 0,C 180,E1 19710.008,E2 19710.008} C_VEL
LIN {X 0,Y 197.777,Z 1293.236,A -85,B 0,C 180,E1 19718.786,E2 19718.786} C_VEL
LIN {X 0,Y 199.502,Z 1286.402,A -85,B 0,C 180,E1 19728.732,E2 19728.732} C_VEL
LIN {X 0,Y 205,Z 1274.131,A -85,B 0,C 180,E1 19738.763,E2 19738.763} C_VEL
LIN {X 0,Y 215.543,Z 1255.33,A -85,B 0,C 180,E1 19748.425,E2 19748.425} C_VEL
LIN {X 0,Y 229.529,Z 1231.334,A -85,B 0,C 180,E1 19756.33,E2 19756.33} C_VEL
LIN {X 0,Y 237.397,Z 1217.84,A -85,B 0,C 180,E1 19759.723,E2 19759.723} C_VEL
LIN {X 0,Y 247.059,Z 1209.713,A -85,B 0,C 180,E1 19762.577,E2 19762.577} C_VEL
LIN {X 0,Y 248.103,Z 1208.672,A -85,B 0,C 180,E1 19763.279,E2 19763.279} C_VEL
LIN {X 0,Y 225.44,Z 1218.723,A -85,B 0,C 180,E1 19772.06,E2 19772.06} C_VEL
LIN {X 0,Y 214.214,Z 1221.888,A -85,B 0,C 180,E1 19779.377,E2 19779.377} C_VEL
LIN {X 0,Y 206.553,Z 1221.54,A -85,B 0,C 180,E1 19787.339,E2 19787.339} C_VEL
LIN {X 0,Y 202.451,Z 1217.227,A -85,B 0,C 180,E1 19795.725,E2 19795.725} C_VEL
LIN {X 0,Y 201.601,Z 1207.106,A -85,B 0,C 180,E1 19805.368,E2 19805.368} C_VEL
LIN {X 0,Y 203.706,Z 1191.814,A -85,B 0,C 180,E1 19814.295,E2 19814.295} C_VEL
LIN {X 0,Y 205.519,Z 1185.14,A -85,B 0,C 180,E1 19817.684,E2 19817.684} C_VEL
LIN {X 0,Y 218.934,Z 1179.577,A -85,B 0,C 180,E1 19824.9,E2 19824.9} C_VEL
LIN {X 0,Y 234.854,Z 1176.773,A -85,B 0,C 180,E1 19832.129,E2 19832.129} C_VEL
LIN {X 0,Y 236.272,Z 1176.161,A -85,B 0,C 180,E1 19832.501,E2 19832.501} C_VEL
LIN {X 0,Y 253.201,Z 1167.643,A -85,B 0,C 180,E1 19836.05,E2 19836.05} C_VEL
LIN {X 0,Y 253.195,Z 1169.535,A -85,B 0,C 180,E1 19836.64,E2 19836.64} C_VEL
LIN {X 0,Y 237.628,Z 1197.346,A -85,B 0,C 180,E1 19841.692,E2 19841.692} C_VEL
LIN {X 0,Y 221.313,Z 1221.895,A -85,B 0,C 180,E1 19848.589,E2 19848.589} C_VEL
LIN {X 0,Y 207.294,Z 1241.027,A -85,B 0,C 180,E1 19857.089,E2 19857.089} C_VEL
LIN {X 0,Y 196.845,Z 1254.966,A -85,B 0,C 180,E1 19867.452,E2 19867.452} C_VEL
LIN {X 0,Y 191.468,Z 1263.032,A -85,B 0,C 180,E1 19878.627,E2 19878.627} C_VEL
LIN {X 0,Y 190.128,Z 1265.641,A -85,B 0,C 180,E1 19889.991,E2 19889.991} C_VEL
LIN {X 0,Y 191.01,Z 1263.904,A -85,B 0,C 180,E1 19899.082,E2 19899.082} C_VEL
LIN {X 0,Y 195.418,Z 1256.996,A -85,B 0,C 180,E1 19910.325,E2 19910.325} C_VEL
LIN {X 0,Y 204.944,Z 1243.941,A -85,B 0,C 180,E1 19921.016,E2 19921.016} C_VEL
LIN {X 0,Y 219.021,Z 1225.005,A -85,B 0,C 180,E1 19930.175,E2 19930.175} C_VEL
LIN {X 0,Y 234.98,Z 1201.401,A -85,B 0,C 180,E1 19937.234,E2 19937.234} C_VEL
LIN {X 0,Y 250.915,Z 1173.756,A -85,B 0,C 180,E1 19942.586,E2 19942.586} C_VEL
LIN {X 0,Y 265.383,Z 1142.282,A -85,B 0,C 180,E1 19946.623,E2 19946.623} C_VEL
LIN {X 0,Y 271.302,Z 1125.754,A -85,B 0,C 180,E1 19948.221,E2 19948.221} C_VEL
LIN {X 0,Y 268.363,Z 1106.853,A -85,B 0,C 180,E1 19953.269,E2 19953.269} C_VEL
LIN {X 0,Y 262.877,Z 1088.141,A -85,B 0,C 180,E1 19959.855,E2 19959.855} C_VEL
LIN {X 0,Y 257.687,Z 1074.889,A -85,B 0,C 180,E1 19966.778,E2 19966.778} C_VEL
LIN {X 0,Y 254.41,Z 1066.318,A -85,B 0,C 180,E1 19974.043,E2 19974.043} C_VEL
LIN {X 0,Y 253.823,Z 1065.605,A -85,B 0,C 180,E1 19982.556,E2 19982.556} C_VEL
LIN {X 0,Y 254.992,Z 1067.727,A -85,B 0,C 180,E1 19986.371,E2 19986.371} C_VEL
LIN {X 0,Y 258.497,Z 1075.489,A -85,B 0,C 180,E1 19992.538,E2 19992.538} C_VEL
LIN {X 0,Y 263.806,Z 1086.634,A -85,B 0,C 180,E1 19998.337,E2 19998.337} C_VEL
LIN {X 0,Y 266.411,Z 1124.309,A -85,B 0,C 180,E1 20005.908,E2 20005.908} C_VEL
LIN {X 0,Y 266.81,Z 1135.176,A -85,B 0,C 180,E1 20008.053,E2 20008.053} C_VEL
LIN {X 0,Y 254.622,Z 1169.178,A -85,B 0,C 180,E1 20011.18,E2 20011.18} C_VEL
LIN {X 0,Y 240.624,Z 1199.577,A -85,B 0,C 180,E1 20015.396,E2 20015.396} C_VEL
LIN {X 0,Y 225.52,Z 1227.316,A -85,B 0,C 180,E1 20021.179,E2 20021.179} C_VEL
LIN {X 0,Y 210.91,Z 1251.356,A -85,B 0,C 180,E1 20028.814,E2 20028.814} C_VEL
LIN {X 0,Y 199.42,Z 1270.244,A -85,B 0,C 180,E1 20038.024,E2 20038.024} C_VEL
LIN {X 0,Y 192.167,Z 1284.573,A -85,B 0,C 180,E1 20049.163,E2 20049.163} C_VEL
LIN {X 0,Y 190.038,Z 1291.528,A -85,B 0,C 180,E1 20058.559,E2 20058.559} C_VEL
LIN {X 0,Y 189.761,Z 1294.094,A -85,B 0,C 180,E1 20065.448,E2 20065.448} C_VEL
LIN {X 0,Y 190.05,Z 1294.656,A -85,B 0,C 180,E1 20070.009,E2 20070.009} C_VEL
LIN {X 0,Y 189.889,Z 1292.627,A -85,B 0,C 180,E1 20079.154,E2 20079.154} C_VEL
LIN {X 0,Y 191.743,Z 1286.059,A -85,B 0,C 180,E1 20089.202,E2 20089.202} C_VEL
LIN {X 0,Y 197.708,Z 1273.731,A -85,B 0,C 180,E1 20099.754,E2 20099.754} C_VEL
LIN {X 0,Y 209.176,Z 1254.709,A -85,B 0,C 180,E1 20109.822,E2 20109.822} C_VEL
LIN {X 0,Y 223.939,Z 1230.716,A -85,B 0,C 180,E1 20117.849,E2 20117.849} C_VEL
LIN {X 0,Y 230.094,Z 1221.234,A -85,B 0,C 180,E1 20120.421,E2 20120.421} C_VEL
LIN {X 0,Y 239.061,Z 1214.147,A -85,B 0,C 180,E1 20123.375,E2 20123.375} C_VEL
LIN {X 0,Y 218.968,Z 1221.573,A -85,B 0,C 180,E1 20131.158,E2 20131.158} C_VEL
LIN {X 0,Y 207.149,Z 1224.087,A -85,B 0,C 180,E1 20138.64,E2 20138.64} C_VEL
LIN {X 0,Y 199.027,Z 1223.178,A -85,B 0,C 180,E1 20146.852,E2 20146.852} C_VEL
LIN {X 0,Y 194.171,Z 1216.508,A -85,B 0,C 180,E1 20157.772,E2 20157.772} C_VEL
LIN {X 0,Y 193.862,Z 1206.179,A -85,B 0,C 180,E1 20166.704,E2 20166.704} C_VEL
LIN {X 0,Y 195.991,Z 1193.052,A -85,B 0,C 180,E1 20174.648,E2 20174.648} C_VEL
LIN {X 0,Y 215.297,Z 1185.315,A -85,B 0,C 180,E1 20185.931,E2 20185.931} C_VEL
LIN {X 0,Y 236.272,Z 1176.161,A -85,B 0,C 180,E1 20192.501,E2 20192.501} C_VEL
LIN {X 0,Y 239.443,Z 1176.495,A -85,B 0,C 180,E1 20193.954,E2 20193.954} C_VEL
LIN {X 0,Y 240.128,Z 1181.017,A -85,B 0,C 180,E1 20195.969,E2 20195.969} C_VEL
LIN {X 0,Y 237.019,Z 1190.315,A -85,B 0,C 180,E1 20198.572,E2 20198.572} C_VEL
LIN {X 0,Y 235.158,Z 1193.598,A -85,B 0,C 180,E1 20199.308,E2 20199.308} C_VEL
LIN {X 0,Y 218.694,Z 1218.083,A -85,B 0,C 180,E1 20205.67,E2 20205.67} C_VEL
LIN {X 0,Y 203.832,Z 1237.619,A -85,B 0,C 180,E1 20213.671,E2 20213.671} C_VEL
LIN {X 0,Y 191.835,Z 1252.615,A -85,B 0,C 180,E1 20223.718,E2 20223.718} C_VEL
LIN {X 0,Y 185.45,Z 1261.089,A -85,B 0,C 180,E1 20233.444,E2 20233.444} C_VEL
LIN {X 0,Y 182.885,Z 1265.032,A -85,B 0,C 180,E1 20241.921,E2 20241.921} C_VEL
LIN {X 0,Y 182.249,Z 1266.242,A -85,B 0,C 180,E1 20249.991,E2 20249.991} C_VEL
LIN {X 0,Y 183.191,Z 1264.509,A -85,B 0,C 180,E1 20259.474,E2 20259.474} C_VEL
LIN {X 0,Y 187.988,Z 1257.602,A -85,B 0,C 180,E1 20271.166,E2 20271.166} C_VEL
LIN {X 0,Y 198.165,Z 1244.548,A -85,B 0,C 180,E1 20282.203,E2 20282.203} C_VEL
LIN {X 0,Y 212.565,Z 1226.161,A -85,B 0,C 180,E1 20291.337,E2 20291.337} C_VEL
LIN {X 0,Y 229.366,Z 1202.451,A -85,B 0,C 180,E1 20298.585,E2 20298.585} C_VEL
